LIN {X 0,Y 105.303,Z 769.102,A -85,B 0,C 180,E1 -26364.249,E2 -26364.249} C_VEL
LIN {X 0,Y 105.299,Z 772.199,A -85,B 0,C 180,E1 -26369.995,E2 -26369.995} C_VEL
LIN {X 0,Y 105.168,Z 773.673,A -85,B 0,C 180,E1 -26373.826,E2 -26373.826} C_VEL
LIN {X 0,Y 105.345,Z 774.732,A -85,B 0,C 180,E1 -26377.662,E2 -26377.662} C_VEL
LIN {X 0,Y 106.79,Z 775.648,A -85,B 0,C 180,E1 -26385.257,E2 -26385.257} C_VEL
LIN {X 0,Y 109.908,Z 775.104,A -85,B 0,C 180,E1 -26392.555,E2 -26392.555} C_VEL
LIN {X 0,Y 112.231,Z 774.277,A -85,B 0,C 180,E1 -26395.992,E2 -26395.992} C_VEL
LIN {X 0,Y 118.036,Z 771.438,A -85,B 0,C 180,E1 -26402.397,E2 -26402.397} C_VEL
LIN {X 0,Y 125.236,Z 766.969,A -85,B 0,C 180,E1 -26408.216,E2 -26408.216} C_VEL
LIN {X 0,Y 131.258,Z 762.539,A -85,B 0,C 180,E1 -26412.006,E2 -26412.006} C_VEL
LIN {X 0,Y 139.26,Z 755.845,A -85,B 0,C 180,E1 -26415.978,E2 -26415.978} C_VEL
LIN {X 0,Y 146.598,Z 748.7,A -85,B 0,C 180,E1 -26419.025,E2 -26419.025} C_VEL
LIN {X 0,Y 154.378,Z 739.924,A -85,B 0,C 180,E1 -26421.742,E2 -26421.742} C_VEL
LIN {X 0,Y 161.875,Z 729.959,A -85,B 0,C 180,E1 -26423.955,E2 -26423.955} C_VEL
LIN {X 0,Y 168.922,Z 718.713,A -85,B 0,C 180,E1 -26425.775,E2 -26425.775} C_VEL
LIN {X 0,Y 174.757,Z 707.532,A -85,B 0,C 180,E1 -26427.081,E2 -26427.081} C_VEL
LIN {X 0,Y 175.208,Z 706.525,A -85,B 0,C 180,E1 -26427.178,E2 -26427.178} C_VEL
LIN {X 0,Y 176.538,Z 703.106,A -85,B 0,C 180,E1 -26427.707,E2 -26427.707} C_VEL
LIN {X 0,Y 179.141,Z 692.574,A -85,B 0,C 180,E1 -26430.31,E2 -26430.31} C_VEL
LIN {X 0,Y 180.193,Z 688.973,A -85,B 0,C 180,E1 -26430.72,E2 -26430.72} C_VEL
LIN {X 0,Y 183.852,Z 675.631,A -85,B 0,C 180,E1 -26431.326,E2 -26431.326} C_VEL
LIN {X 0,Y 185.48,Z 666.767,A -85,B 0,C 180,E1 -26431.645,E2 -26431.645} C_VEL
LIN {X 0,Y 184.736,Z 662.719,A -85,B 0,C 180,E1 -26434.358,E2 -26434.358} C_VEL
LIN {X 0,Y 184.119,Z 659.45,A -85,B 0,C 180,E1 -26438.256,E2 -26438.256} C_VEL
LIN {X 0,Y 184.228,Z 658.963,A -85,B 0,C 180,E1 -26442.487,E2 -26442.487} C_VEL
LIN {X 0,Y 185.103,Z 661.189,A -85,B 0,C 180,E1 -26446.452,E2 -26446.452} C_VEL
LIN {X 0,Y 185.885,Z 663.628,A -85,B 0,C 180,E1 -26448.675,E2 -26448.675} C_VEL
LIN {X 0,Y 183.18,Z 677.331,A -85,B 0,C 180,E1 -26449.199,E2 -26449.199} C_VEL
LIN {X 0,Y 179.514,Z 689.858,A -85,B 0,C 180,E1 -26449.939,E2 -26449.939} C_VEL
LIN {X 0,Y 174.557,Z 702.362,A -85,B 0,C 180,E1 -26451.004,E2 -26451.004} C_VEL
LIN {X 0,Y 169.094,Z 713.244,A -85,B 0,C 180,E1 -26452.244,E2 -26452.244} C_VEL
LIN {X 0,Y 162.575,Z 723.845,A -85,B 0,C 180,E1 -26453.826,E2 -26453.826} C_VEL
LIN {X 0,Y 154.993,Z 734.01,A -85,B 0,C 180,E1 -26455.944,E2 -26455.944} C_VEL
LIN {X 0,Y 147.643,Z 742.315,A -85,B 0,C 180,E1 -26458.279,E2 -26458.279} C_VEL
LIN {X 0,Y 139.13,Z 750.499,A -85,B 0,C 180,E1 -26461.412,E2 -26461.412} C_VEL
LIN {X 0,Y 130.939,Z 757.072,A -85,B 0,C 180,E1 -26465.062,E2 -26465.062} C_VEL
LIN {X 0,Y 122.214,Z 762.916,A -85,B 0,C 180,E1 -26469.932,E2 -26469.932} C_VEL
LIN {X 0,Y 116.026,Z 766.288,A -85,B 0,C 180,E1 -26474.287,E2 -26474.287} C_VEL
LIN {X 0,Y 111.192,Z 768.427,A -85,B 0,C 180,E1 -26478.56,E2 -26478.56} C_VEL
LIN {X 0,Y 106.98,Z 769.842,A -85,B 0,C 180,E1 -26483.212,E2 -26483.212} C_VEL
LIN {X 0,Y 103.362,Z 770.554,A -85,B 0,C 180,E1 -26488.419,E2 -26488.419} C_VEL
LIN {X 0,Y 100.652,Z 770.454,A -85,B 0,C 180,E1 -26493.956,E2 -26493.956} C_VEL
LIN {X 0,Y 98.728,Z 769.526,A -85,B 0,C 180,E1 -26499.839,E2 -26499.839} C_VEL
LIN {X 0,Y 97.648,Z 767.699,A -85,B 0,C 180,E1 -26506.029,E2 -26506.029} C_VEL
LIN {X 0,Y 97.544,Z 764.862,A -85,B 0,C 180,E1 -26512.42,E2 -26512.42} C_VEL
LIN {X 0,Y 98.341,Z 760.757,A -85,B 0,C 180,E1 -26519.043,E2 -26519.043} C_VEL
LIN {X 0,Y 100.087,Z 755.004,A -85,B 0,C 180,E1 -26525.897,E2 -26525.897} C_VEL
LIN {X 0,Y 102.312,Z 748.886,A -85,B 0,C 180,E1 -26531.427,E2 -26531.427} C_VEL
LIN {X 0,Y 105.063,Z 741.752,A -85,B 0,C 180,E1 -26536.466,E2 -26536.466} C_VEL
LIN {X 0,Y 108.553,Z 733.143,A -85,B 0,C 180,E1 -26541.16,E2 -26541.16} C_VEL
LIN {X 0,Y 112.175,Z 723.535,A -85,B 0,C 180,E1 -26545.211,E2 -26545.211} C_VEL
LIN {X 0,Y 116.013,Z 712.64,A -85,B 0,C 180,E1 -26548.703,E2 -26548.703} C_VEL
LIN {X 0,Y 119.515,Z 700.829,A -85,B 0,C 180,E1 -26551.54,E2 -26551.54} C_VEL
LIN {X 0,Y 122.584,Z 688.566,A -85,B 0,C 180,E1 -26553.703,E2 -26553.703} C_VEL
LIN {X 0,Y 125.058,Z 675.36,A -85,B 0,C 180,E1 -26555.345,E2 -26555.345} C_VEL
LIN {X 0,Y 126.899,Z 661.316,A -85,B 0,C 180,E1 -26556.426,E2 -26556.426} C_VEL
LIN {X 0,Y 130.052,Z 624.131,A -85,B 0,C 180,E1 -26558.464,E2 -26558.464} C_VEL
LIN {X 0,Y 123.711,Z 608.885,A -85,B 0,C 180,E1 -26561.983,E2 -26561.983} C_VEL
LIN {X 0,Y 115.972,Z 594.893,A -85,B 0,C 180,E1 -26566.547,E2 -26566.547} C_VEL
LIN {X 0,Y 110.04,Z 585.76,A -85,B 0,C 180,E1 -26570.479,E2 -26570.479} C_VEL
LIN {X 0,Y 107.393,Z 581.803,A -85,B 0,C 180,E1 -26572.446,E2 -26572.446} C_VEL
LIN {X 0,Y 104.798,Z 578.322,A -85,B 0,C 180,E1 -26574.502,E2 -26574.502} C_VEL
LIN {X 0,Y 104.228,Z 577.151,A -85,B 0,C 180,E1 -26575.032,E2 -26575.032} C_VEL
LIN {X 0,Y 102,Z 575.216,A -85,B 0,C 180,E1 -26576.806,E2 -26576.806} C_VEL
LIN {X 0,Y 100.845,Z 572.761,A -85,B 0,C 180,E1 -26577.978,E2 -26577.978} C_VEL
LIN {X 0,Y 100.663,Z 571.949,A -85,B 0,C 180,E1 -26578.344,E2 -26578.344} C_VEL
LIN {X 0,Y 100.666,Z 571.937,A -85,B 0,C 180,E1 -26583.96,E2 -26583.96} C_VEL
LIN {X 0,Y 100.643,Z 571.931,A -85,B 0,C 180,E1 -26589.816,E2 -26589.816} C_VEL
LIN {X 0,Y 100.652,Z 571.948,A -85,B 0,C 180,E1 -26595.716,E2 -26595.716} C_VEL
LIN {X 0,Y 100.631,Z 571.925,A -85,B 0,C 180,E1 -26601.059,E2 -26601.059} C_VEL
LIN {X 0,Y 100.695,Z 571.94,A -85,B 0,C 180,E1 -26606.891,E2 -26606.891} C_VEL
LIN {X 0,Y 100.794,Z 571.925,A -85,B 0,C 180,E1 -26615.271,E2 -26615.271} C_VEL
LIN {X 0,Y 100.816,Z 571.915,A -85,B 0,C 180,E1 -26619.603,E2 -26619.603} C_VEL
LIN {X 0,Y 101.168,Z 571.883,A -85,B 0,C 180,E1 -26627.973,E2 -26627.973} C_VEL
LIN {X 0,Y 101.251,Z 571.851,A -85,B 0,C 180,E1 -26632.022,E2 -26632.022} C_VEL
LIN {X 0,Y 101.876,Z 571.793,A -85,B 0,C 180,E1 -26640.002,E2 -26640.002} C_VEL
LIN {X 0,Y 101.285,Z 571.868,A -85,B 0,C 180,E1 -26647.979,E2 -26647.979} C_VEL
LIN {X 0,Y 101.123,Z 571.872,A -85,B 0,C 180,E1 -26653.324,E2 -26653.324} C_VEL
LIN {X 0,Y 100.824,Z 571.887,A -85,B 0,C 180,E1 -26661.334,E2 -26661.334} C_VEL
LIN {X 0,Y 101.671,Z 574.415,A -85,B 0,C 180,E1 -26662.347,E2 -26662.347} C_VEL
LIN {X 0,Y 103.856,Z 576.845,A -85,B 0,C 180,E1 -26664.223,E2 -26664.223} C_VEL
LIN {X 0,Y 106.376,Z 580.87,A -85,B 0,C 180,E1 -26666.354,E2 -26666.354} C_VEL
LIN {X 0,Y 107.782,Z 582.765,A -85,B 0,C 180,E1 -26667.423,E2 -26667.423} C_VEL
LIN {X 0,Y 112.491,Z 589.94,A -85,B 0,C 180,E1 -26670.767,E2 -26670.767} C_VEL
LIN {X 0,Y 118.61,Z 600.466,A -85,B 0,C 180,E1 -26674.709,E2 -26674.709} C_VEL
LIN {X 0,Y 122.562,Z 609.707,A -85,B 0,C 180,E1 -26677.165,E2 -26677.165} C_VEL
LIN {X 0,Y 126.766,Z 621.513,A -85,B 0,C 180,E1 -26679.728,E2 -26679.728} C_VEL
LIN {X 0,Y 129.782,Z 631.148,A -85,B 0,C 180,E1 -26681.535,E2 -26681.535} C_VEL
LIN {X 0,Y 126.025,Z 673.787,A -85,B 0,C 180,E1 -26683.961,E2 -26683.961} C_VEL
LIN {X 0,Y 123.841,Z 687.25,A -85,B 0,C 180,E1 -26685.241,E2 -26685.241} C_VEL
LIN {X 0,Y 121.065,Z 699.593,A -85,B 0,C 180,E1 -26686.986,E2 -26686.986} C_VEL
LIN {X 0,Y 117.605,Z 711.948,A -85,B 0,C 180,E1 -26689.461,E2 -26689.461} C_VEL
LIN {X 0,Y 113.967,Z 723.108,A -85,B 0,C 180,E1 -26692.479,E2 -26692.479} C_VEL
LIN {X 0,Y 110.055,Z 733.645,A -85,B 0,C 180,E1 -26696.283,E2 -26696.283} C_VEL
LIN {X 0,Y 106.01,Z 743.969,A -85,B 0,C 180,E1 -26701.267,E2 -26701.267} C_VEL
LIN {X 0,Y 102.656,Z 752.512,A -85,B 0,C 180,E1 -26706.812,E2 -26706.812} C_VEL
LIN {X 0,Y 100.226,Z 759.339,A -85,B 0,C 180,E1 -26712.656,E2 -26712.656} C_VEL
LIN {X 0,Y 98.654,Z 765.567,A -85,B 0,C 180,E1 -26719.735,E2 -26719.735} C_VEL
LIN {X 0,Y 98.19,Z 769.554,A -85,B 0,C 180,E1 -26725.89,E2 -26725.89} C_VEL
LIN {X 0,Y 98.234,Z 771.574,A -85,B 0,C 180,E1 -26729.994,E2 -26729.994} C_VEL
LIN {X 0,Y 98.094,Z 773.12,A -85,B 0,C 180,E1 -26734.103,E2 -26734.103} C_VEL
LIN {X 0,Y 98.897,Z 775.038,A -85,B 0,C 180,E1 -26742.303,E2 -26742.303} C_VEL
LIN {X 0,Y 101.407,Z 775.387,A -85,B 0,C 180,E1 -26750.269,E2 -26750.269} C_VEL
LIN {X 0,Y 105.888,Z 774.285,A -85,B 0,C 180,E1 -26757.678,E2 -26757.678} C_VEL
LIN {X 0,Y 112.1,Z 771.687,A -85,B 0,C 180,E1 -26764.343,E2 -26764.343} C_VEL
LIN {X 0,Y 119.646,Z 767.467,A -85,B 0,C 180,E1 -26770.245,E2 -26770.245} C_VEL
LIN {X 0,Y 126.112,Z 763.193,A -85,B 0,C 180,E1 -26774.148,E2 -26774.148} C_VEL
LIN {X 0,Y 134.473,Z 756.819,A -85,B 0,C 180,E1 -26778.131,E2 -26778.131} C_VEL
LIN {X 0,Y 142.121,Z 749.947,A -85,B 0,C 180,E1 -26781.149,E2 -26781.149} C_VEL
LIN {X 0,Y 150.176,Z 741.472,A -85,B 0,C 180,E1 -26783.823,E2 -26783.823} C_VEL
LIN {X 0,Y 157.178,Z 732.942,A -85,B 0,C 180,E1 -26785.805,E2 -26785.805} C_VEL
LIN {X 0,Y 164.413,Z 722.56,A -85,B 0,C 180,E1 -26787.583,E2 -26787.583} C_VEL
LIN {X 0,Y 171.098,Z 710.87,A -85,B 0,C 180,E1 -26789.025,E2 -26789.025} C_VEL
LIN {X 0,Y 176.407,Z 699.321,A -85,B 0,C 180,E1 -26790.048,E2 -26790.048} C_VEL
LIN {X 0,Y 180.193,Z 688.973,A -85,B 0,C 180,E1 -26790.72,E2 -26790.72} C_VEL
LIN {X 0,Y 182.064,Z 682.31,A -85,B 0,C 180,E1 -26791.231,E2 -26791.231} C_VEL
LIN {X 0,Y 183.034,Z 677.264,A -85,B 0,C 180,E1 -26791.947,E2 -26791.947} C_VEL
LIN {X 0,Y 183.418,Z 673.974,A -85,B 0,C 180,E1 -26792.699,E2 -26792.699} C_VEL
LIN {X 0,Y 183.499,Z 671.379,A -85,B 0,C 180,E1 -26793.666,E2 -26793.666} C_VEL
LIN {X 0,Y 183.46,Z 670.748,A -85,B 0,C 180,E1 -26794.038,E2 -26794.038} C_VEL
LIN {X 0,Y 183.185,Z 668.656,A -85,B 0,C 180,E1 -26795.704,E2 -26795.704} C_VEL
LIN {X 0,Y 182.935,Z 666.303,A -85,B 0,C 180,E1 -26798.908,E2 -26798.908} C_VEL
LIN {X 0,Y 183.127,Z 666.057,A -85,B 0,C 180,E1 -26802.726,E2 -26802.726} C_VEL
LIN {X 0,Y 183.726,Z 668.003,A -85,B 0,C 180,E1 -26805.967,E2 -26805.967} C_VEL
LIN {X 0,Y 183.867,Z 668.892,A -85,B 0,C 180,E1 -26806.677,E2 -26806.677} C_VEL
LIN {X 0,Y 180.525,Z 682.697,A -85,B 0,C 180,E1 -26807.255,E2 -26807.255} C_VEL
LIN {X 0,Y 176.457,Z 694.617,A -85,B 0,C 180,E1 -26808.019,E2 -26808.019} C_VEL
LIN {X 0,Y 170.967,Z 706.812,A -85,B 0,C 180,E1 -26809.11,E2 -26809.11} C_VEL
LIN {X 0,Y 164.778,Z 717.747,A -85,B 0,C 180,E1 -26810.431,E2 -26810.431} C_VEL
LIN {X 0,Y 158.017,Z 727.658,A -85,B 0,C 180,E1 -26812.016,E2 -26812.016} C_VEL
LIN {X 0,Y 150.126,Z 737.27,A -85,B 0,C 180,E1 -26814.098,E2 -26814.098} C_VEL
LIN {X 0,Y 142.587,Z 745.015,A -85,B 0,C 180,E1 -26816.403,E2 -26816.403} C_VEL
LIN {X 0,Y 133.524,Z 752.841,A -85,B 0,C 180,E1 -26819.617,E2 -26819.617} C_VEL
LIN {X 0,Y 125.3,Z 758.814,A -85,B 0,C 180,E1 -26823.214,E2 -26823.214} C_VEL
LIN {X 0,Y 116.21,Z 764.188,A -85,B 0,C 180,E1 -26828.147,E2 -26828.147} C_VEL
LIN {X 0,Y 108.475,Z 767.805,A -85,B 0,C 180,E1 -26833.654,E2 -26833.654} C_VEL
LIN {X 0,Y 101.706,Z 770.024,A -85,B 0,C 180,E1 -26840.21,E2 -26840.21} C_VEL
LIN {X 0,Y 97.606,Z 770.773,A -85,B 0,C 180,E1 -26845.594,E2 -26845.594} C_VEL
LIN {X 0,Y 93.331,Z 770.407,A -85,B 0,C 180,E1 -26854.085,E2 -26854.085} C_VEL
LIN {X 0,Y 91.54,Z 769.325,A -85,B 0,C 180,E1 -26859.858,E2 -26859.858} C_VEL
LIN {X 0,Y 90.414,Z 766.441,A -85,B 0,C 180,E1 -26868.538,E2 -26868.538} C_VEL
LIN {X 0,Y 90.943,Z 761.922,A -85,B 0,C 180,E1 -26877.259,E2 -26877.259} C_VEL
LIN {X 0,Y 92.41,Z 756.802,A -85,B 0,C 180,E1 -26884.25,E2 -26884.25} C_VEL
LIN {X 0,Y 94.536,Z 750.833,A -85,B 0,C 180,E1 -26890.464,E2 -26890.464} C_VEL
LIN {X 0,Y 97.596,Z 743.305,A -85,B 0,C 180,E1 -26896.471,E2 -26896.471} C_VEL
LIN {X 0,Y 101.499,Z 734.024,A -85,B 0,C 180,E1 -26902.046,E2 -26902.046} C_VEL
LIN {X 0,Y 105.598,Z 723.772,A -85,B 0,C 180,E1 -26906.639,E2 -26906.639} C_VEL
LIN {X 0,Y 109.721,Z 712.599,A -85,B 0,C 180,E1 -26910.377,E2 -26910.377} C_VEL
LIN {X 0,Y 113.283,Z 701.181,A -85,B 0,C 180,E1 -26913.223,E2 -26913.223} C_VEL
LIN {X 0,Y 116.772,Z 687.915,A -85,B 0,C 180,E1 -26915.617,E2 -26915.617} C_VEL
LIN {X 0,Y 119.258,Z 674.646,A -85,B 0,C 180,E1 -26917.282,E2 -26917.282} C_VEL
LIN {X 0,Y 121.047,Z 661.623,A -85,B 0,C 180,E1 -26918.288,E2 -26918.288} C_VEL
LIN {X 0,Y 124.269,Z 626.1,A -85,B 0,C 180,E1 -26920.271,E2 -26920.271} C_VEL
LIN {X 0,Y 118.738,Z 612.717,A -85,B 0,C 180,E1 -26923.581,E2 -26923.581} C_VEL
LIN {X 0,Y 111.803,Z 599.793,A -85,B 0,C 180,E1 -26928.036,E2 -26928.036} C_VEL
LIN {X 0,Y 106.071,Z 590.815,A -85,B 0,C 180,E1 -26932.154,E2 -26932.154} C_VEL
LIN {X 0,Y 102.725,Z 585.931,A -85,B 0,C 180,E1 -26934.902,E2 -26934.902} C_VEL
LIN {X 0,Y 100.659,Z 582.889,A -85,B 0,C 180,E1 -26936.715,E2 -26936.715} C_VEL
LIN {X 0,Y 98.196,Z 579.989,A -85,B 0,C 180,E1 -26938.969,E2 -26938.969} C_VEL
LIN {X 0,Y 97.32,Z 578.208,A -85,B 0,C 180,E1 -26939.94,E2 -26939.94} C_VEL
LIN {X 0,Y 94.941,Z 576.16,A -85,B 0,C 180,E1 -26942.331,E2 -26942.331} C_VEL
LIN {X 0,Y 93.694,Z 573.326,A -85,B 0,C 180,E1 -26944.003,E2 -26944.003} C_VEL
LIN {X 0,Y 93.595,Z 572.819,A -85,B 0,C 180,E1 -26944.315,E2 -26944.315} C_VEL
LIN {X 0,Y 93.537,Z 572.819,A -85,B 0,C 180,E1 -26952.557,E2 -26952.557} C_VEL
LIN {X 0,Y 93.54,Z 572.813,A -85,B 0,C 180,E1 -26958.715,E2 -26958.715} C_VEL
LIN {X 0,Y 93.592,Z 572.828,A -85,B 0,C 180,E1 -26965.701,E2 -26965.701} C_VEL
LIN {X 0,Y 93.675,Z 572.802,A -85,B 0,C 180,E1 -26974.211,E2 -26974.211} C_VEL
LIN {X 0,Y 93.696,Z 572.811,A -85,B 0,C 180,E1 -26977.976,E2 -26977.976} C_VEL
LIN {X 0,Y 94.077,Z 572.764,A -85,B 0,C 180,E1 -26987.051,E2 -26987.051} C_VEL
LIN {X 0,Y 94.185,Z 572.734,A -85,B 0,C 180,E1 -26991.419,E2 -26991.419} C_VEL
LIN {X 0,Y 94.801,Z 572.674,A -85,B 0,C 180,E1 -27000.002,E2 -27000.002} C_VEL
LIN {X 0,Y 94.218,Z 572.75,A -85,B 0,C 180,E1 -27008.582,E2 -27008.582} C_VEL
LIN {X 0,Y 94.044,Z 572.754,A -85,B 0,C 180,E1 -27013.689,E2 -27013.689} C_VEL
LIN {X 0,Y 93.907,Z 572.785,A -85,B 0,C 180,E1 -27015.639,E2 -27015.639} C_VEL
LIN {X 0,Y 94.721,Z 575.446,A -85,B 0,C 180,E1 -27016.858,E2 -27016.858} C_VEL
LIN {X 0,Y 96.625,Z 577.643,A -85,B 0,C 180,E1 -27018.882,E2 -27018.882} C_VEL
LIN {X 0,Y 97.639,Z 578.51,A -85,B 0,C 180,E1 -27019.857,E2 -27019.857} C_VEL
LIN {X 0,Y 99.718,Z 581.799,A -85,B 0,C 180,E1 -27021.942,E2 -27021.942} C_VEL
LIN {X 0,Y 100.982,Z 583.43,A -85,B 0,C 180,E1 -27023.083,E2 -27023.083} C_VEL
LIN {X 0,Y 103.649,Z 587.259,A -85,B 0,C 180,E1 -27025.423,E2 -27025.423} C_VEL
LIN {X 0,Y 109.031,Z 596,A -85,B 0,C 180,E1 -27029.64,E2 -27029.64} C_VEL
LIN {X 0,Y 114.357,Z 605.405,A -85,B 0,C 180,E1 -27033.293,E2 -27033.293} C_VEL
LIN {X 0,Y 118.618,Z 616.25,A -85,B 0,C 180,E1 -27036.217,E2 -27036.217} C_VEL
LIN {X 0,Y 122.728,Z 628.647,A -85,B 0,C 180,E1 -27038.914,E2 -27038.914} C_VEL
LIN {X 0,Y 123.981,Z 632.936,A -85,B 0,C 180,E1 -27039.732,E2 -27039.732} C_VEL
LIN {X 0,Y 120.183,Z 673.625,A -85,B 0,C 180,E1 -27042.097,E2 -27042.097} C_VEL
LIN {X 0,Y 117.913,Z 687.04,A -85,B 0,C 180,E1 -27043.407,E2 -27043.407} C_VEL
LIN {X 0,Y 114.895,Z 699.847,A -85,B 0,C 180,E1 -27045.29,E2 -27045.29} C_VEL
LIN {X 0,Y 111.273,Z 712.077,A -85,B 0,C 180,E1 -27047.843,E2 -27047.843} C_VEL
LIN {X 0,Y 107.478,Z 723.156,A -85,B 0,C 180,E1 -27050.989,E2 -27050.989} C_VEL
LIN {X 0,Y 103.561,Z 733.174,A -85,B 0,C 180,E1 -27054.779,E2 -27054.779} C_VEL
LIN {X 0,Y 99.795,Z 742.237,A -85,B 0,C 180,E1 -27059.291,E2 -27059.291} C_VEL
LIN {X 0,Y 96.156,Z 751.117,A -85,B 0,C 180,E1 -27065.142,E2 -27065.142} C_VEL
LIN {X 0,Y 93.433,Z 758.164,A -85,B 0,C 180,E1 -27071.35,E2 -27071.35} C_VEL
LIN {X 0,Y 92.05,Z 762.964,A -85,B 0,C 180,E1 -27076.753,E2 -27076.753} C_VEL
LIN {X 0,Y 91.215,Z 767.526,A -85,B 0,C 180,E1 -27083.357,E2 -27083.357} C_VEL
LIN {X 0,Y 91.159,Z 770.934,A -85,B 0,C 180,E1 -27089.994,E2 -27089.994} C_VEL
LIN {X 0,Y 91.033,Z 772.568,A -85,B 0,C 180,E1 -27094.421,E2 -27094.421} C_VEL
LIN {X 0,Y 91.972,Z 774.634,A -85,B 0,C 180,E1 -27103.246,E2 -27103.246} C_VEL
LIN {X 0,Y 94.744,Z 775.214,A -85,B 0,C 180,E1 -27111.764,E2 -27111.764} C_VEL
LIN {X 0,Y 99.651,Z 774.282,A -85,B 0,C 180,E1 -27119.576,E2 -27119.576} C_VEL
LIN {X 0,Y 106.313,Z 771.897,A -85,B 0,C 180,E1 -27126.503,E2 -27126.503} C_VEL
LIN {X 0,Y 113.657,Z 768.333,A -85,B 0,C 180,E1 -27132.093,E2 -27132.093} C_VEL
LIN {X 0,Y 121.159,Z 763.868,A -85,B 0,C 180,E1 -27136.468,E2 -27136.468} C_VEL
LIN {X 0,Y 128.634,Z 758.696,A -85,B 0,C 180,E1 -27139.891,E2 -27139.891} C_VEL
LIN {X 0,Y 135.135,Z 753.511,A -85,B 0,C 180,E1 -27142.47,E2 -27142.47} C_VEL
LIN {X 0,Y 143.375,Z 745.974,A -85,B 0,C 180,E1 -27145.183,E2 -27145.183} C_VEL
LIN {X 0,Y 151.932,Z 736.663,A -85,B 0,C 180,E1 -27147.579,E2 -27147.579} C_VEL
LIN {X 0,Y 159.326,Z 727.15,A -85,B 0,C 180,E1 -27149.327,E2 -27149.327} C_VEL
LIN {X 0,Y 166.141,Z 716.698,A -85,B 0,C 180,E1 -27150.739,E2 -27150.739} C_VEL
LIN {X 0,Y 172.313,Z 705.095,A -85,B 0,C 180,E1 -27151.877,E2 -27151.877} C_VEL
LIN {X 0,Y 177.442,Z 692.926,A -85,B 0,C 180,E1 -27152.736,E2 -27152.736} C_VEL
LIN {X 0,Y 181.554,Z 679.917,A -85,B 0,C 180,E1 -27153.348,E2 -27153.348} C_VEL
LIN {X 0,Y 183.521,Z 671.13,A -85,B 0,C 180,E1 -27153.73,E2 -27153.73} C_VEL
LIN {X 0,Y 183.46,Z 670.748,A -85,B 0,C 180,E1 -27154.038,E2 -27154.038} C_VEL
LIN {X 0,Y 183.232,Z 669.591,A -85,B 0,C 180,E1 -27155.204,E2 -27155.204} C_VEL
LIN {X 0,Y 182.925,Z 669.204,A -85,B 0,C 180,E1 -27156.423,E2 -27156.423} C_VEL
LIN {X 0,Y 182.431,Z 669.68,A -85,B 0,C 180,E1 -27158.284,E2 -27158.284} C_VEL
LIN {X 0,Y 181.8,Z 673.828,A -85,B 0,C 180,E1 -27163.994,E2 -27163.994} C_VEL
LIN {X 0,Y 181.888,Z 674.163,A -85,B 0,C 180,E1 -27164.65,E2 -27164.65} C_VEL
LIN {X 0,Y 178.077,Z 687.429,A -85,B 0,C 180,E1 -27165.248,E2 -27165.248} C_VEL
LIN {X 0,Y 173.312,Z 699.666,A -85,B 0,C 180,E1 -27166.1,E2 -27166.1} C_VEL
LIN {X 0,Y 167.586,Z 711.035,A -85,B 0,C 180,E1 -27167.151,E2 -27167.151} C_VEL
LIN {X 0,Y 160.432,Z 722.36,A -85,B 0,C 180,E1 -27168.552,E2 -27168.552} C_VEL
LIN {X 0,Y 152.361,Z 732.83,A -85,B 0,C 180,E1 -27170.366,E2 -27170.366} C_VEL
LIN {X 0,Y 143.363,Z 742.363,A -85,B 0,C 180,E1 -27172.713,E2 -27172.713} C_VEL
LIN {X 0,Y 133.917,Z 750.714,A -85,B 0,C 180,E1 -27175.59,E2 -27175.59} C_VEL
LIN {X 0,Y 126.551,Z 756.163,A -85,B 0,C 180,E1 -27178.27,E2 -27178.27} C_VEL
LIN {X 0,Y 119.496,Z 760.625,A -85,B 0,C 180,E1 -27181.308,E2 -27181.308} C_VEL
LIN {X 0,Y 110.327,Z 765.42,A -85,B 0,C 180,E1 -27186.165,E2 -27186.165} C_VEL
LIN {X 0,Y 102.121,Z 768.687,A -85,B 0,C 180,E1 -27191.913,E2 -27191.913} C_VEL
LIN {X 0,Y 95.925,Z 770.391,A -85,B 0,C 180,E1 -27197.761,E2 -27197.761} C_VEL
LIN {X 0,Y 91.653,Z 771.015,A -85,B 0,C 180,E1 -27203.066,E2 -27203.066} C_VEL
LIN {X 0,Y 88.244,Z 770.918,A -85,B 0,C 180,E1 -27208.843,E2 -27208.843} C_VEL
LIN {X 0,Y 85.729,Z 770.107,A -85,B 0,C 180,E1 -27215.017,E2 -27215.017} C_VEL
LIN {X 0,Y 83.928,Z 768.41,A -85,B 0,C 180,E1 -27222.056,E2 -27222.056} C_VEL
LIN {X 0,Y 83.314,Z 765.764,A -85,B 0,C 180,E1 -27229.389,E2 -27229.389} C_VEL
LIN {X 0,Y 83.787,Z 761.936,A -85,B 0,C 180,E1 -27237.008,E2 -27237.008} C_VEL
LIN {X 0,Y 85.381,Z 756.557,A -85,B 0,C 180,E1 -27244.877,E2 -27244.877} C_VEL
LIN {X 0,Y 87.541,Z 750.8,A -85,B 0,C 180,E1 -27251.276,E2 -27251.276} C_VEL
LIN {X 0,Y 90.724,Z 743.376,A -85,B 0,C 180,E1 -27257.591,E2 -27257.591} C_VEL
LIN {X 0,Y 94.523,Z 734.874,A -85,B 0,C 180,E1 -27263.067,E2 -27263.067} C_VEL
LIN {X 0,Y 98.472,Z 725.496,A -85,B 0,C 180,E1 -27267.632,E2 -27267.632} C_VEL
LIN {X 0,Y 102.6,Z 714.998,A -85,B 0,C 180,E1 -27271.478,E2 -27271.478} C_VEL
LIN {X 0,Y 106.341,Z 704.212,A -85,B 0,C 180,E1 -27274.452,E2 -27274.452} C_VEL
LIN {X 0,Y 109.756,Z 692.262,A -85,B 0,C 180,E1 -27276.901,E2 -27276.901} C_VEL
LIN {X 0,Y 112.679,Z 679.249,A -85,B 0,C 180,E1 -27278.778,E2 -27278.778} C_VEL
LIN {X 0,Y 114.73,Z 666.76,A -85,B 0,C 180,E1 -27279.973,E2 -27279.973} C_VEL
LIN {X 0,Y 118.528,Z 628.194,A -85,B 0,C 180,E1 -27282.205,E2 -27282.205} C_VEL
LIN {X 0,Y 114.105,Z 617.066,A -85,B 0,C 180,E1 -27285.155,E2 -27285.155} C_VEL
LIN {X 0,Y 107.451,Z 604.295,A -85,B 0,C 180,E1 -27289.791,E2 -27289.791} C_VEL
LIN {X 0,Y 101.928,Z 595.485,A -85,B 0,C 180,E1 -27294.189,E2 -27294.189} C_VEL
LIN {X 0,Y 97.589,Z 588.871,A -85,B 0,C 180,E1 -27298.146,E2 -27298.146} C_VEL
LIN {X 0,Y 94.902,Z 585.392,A -85,B 0,C 180,E1 -27300.88,E2 -27300.88} C_VEL
LIN {X 0,Y 94.09,Z 584.155,A -85,B 0,C 180,E1 -27301.802,E2 -27301.802} C_VEL
LIN {X 0,Y 91.705,Z 581.35,A -85,B 0,C 180,E1 -27304.605,E2 -27304.605} C_VEL
LIN {X 0,Y 90.646,Z 579.321,A -85,B 0,C 180,E1 -27306.087,E2 -27306.087} C_VEL
LIN {X 0,Y 88.114,Z 577.476,A -85,B 0,C 180,E1 -27309.386,E2 -27309.386} C_VEL
LIN {X 0,Y 86.79,Z 575.014,A -85,B 0,C 180,E1 -27311.712,E2 -27311.712} C_VEL
LIN {X 0,Y 86.501,Z 573.694,A -85,B 0,C 180,E1 -27312.513,E2 -27312.513} C_VEL
LIN {X 0,Y 86.461,Z 573.69,A -85,B 0,C 180,E1 -27319.441,E2 -27319.441} C_VEL
LIN {X 0,Y 86.535,Z 573.706,A -85,B 0,C 180,E1 -27325.357,E2 -27325.357} C_VEL
LIN {X 0,Y 86.589,Z 573.675,A -85,B 0,C 180,E1 -27333.243,E2 -27333.243} C_VEL
LIN {X 0,Y 86.638,Z 573.666,A -85,B 0,C 180,E1 -27341.069,E2 -27341.069} C_VEL
LIN {X 0,Y 86.94,Z 573.643,A -85,B 0,C 180,E1 -27345.968,E2 -27345.968} C_VEL
LIN {X 0,Y 87.094,Z 573.622,A -85,B 0,C 180,E1 -27350.715,E2 -27350.715} C_VEL
LIN {X 0,Y 87.728,Z 573.555,A -85,B 0,C 180,E1 -27360.002,E2 -27360.002} C_VEL
LIN {X 0,Y 87.156,Z 573.634,A -85,B 0,C 180,E1 -27367.969,E2 -27367.969} C_VEL
LIN {X 0,Y 88.044,Z 576.363,A -85,B 0,C 180,E1 -27369.768,E2 -27369.768} C_VEL
LIN {X 0,Y 89.827,Z 578.433,A -85,B 0,C 180,E1 -27372.346,E2 -27372.346} C_VEL
LIN {X 0,Y 91.023,Z 579.404,A -85,B 0,C 180,E1 -27373.868,E2 -27373.868} C_VEL
LIN {X 0,Y 92.772,Z 582.639,A -85,B 0,C 180,E1 -27376.224,E2 -27376.224} C_VEL
LIN {X 0,Y 94.81,Z 584.857,A -85,B 0,C 180,E1 -27378.453,E2 -27378.453} C_VEL
LIN {X 0,Y 98.123,Z 589.876,A -85,B 0,C 180,E1 -27381.901,E2 -27381.901} C_VEL
LIN {X 0,Y 102.632,Z 596.778,A -85,B 0,C 180,E1 -27385.972,E2 -27385.972} C_VEL
LIN {X 0,Y 108.919,Z 607.942,A -85,B 0,C 180,E1 -27390.903,E2 -27390.903} C_VEL
LIN {X 0,Y 111.04,Z 612.609,A -85,B 0,C 180,E1 -27392.454,E2 -27392.454} C_VEL
LIN {X 0,Y 115.67,Z 625.814,A -85,B 0,C 180,E1 -27395.913,E2 -27395.913} C_VEL
LIN {X 0,Y 118.175,Z 634.265,A -85,B 0,C 180,E1 -27397.729,E2 -27397.729} C_VEL
LIN {X 0,Y 114.52,Z 672.517,A -85,B 0,C 180,E1 -27400.015,E2 -27400.015} C_VEL
LIN {X 0,Y 112.25,Z 685.699,A -85,B 0,C 180,E1 -27401.288,E2 -27401.288} C_VEL
LIN {X 0,Y 109.368,Z 697.803,A -85,B 0,C 180,E1 -27403.026,E2 -27403.026} C_VEL
LIN {X 0,Y 106.113,Z 708.916,A -85,B 0,C 180,E1 -27405.268,E2 -27405.268} C_VEL
LIN {X 0,Y 102.021,Z 720.507,A -85,B 0,C 180,E1 -27408.46,E2 -27408.46} C_VEL
LIN {X 0,Y 97.426,Z 731.977,A -85,B 0,C 180,E1 -27412.773,E2 -27412.773} C_VEL
LIN {X 0,Y 92.998,Z 742.121,A -85,B 0,C 180,E1 -27418.055,E2 -27418.055} C_VEL
LIN {X 0,Y 89.162,Z 750.981,A -85,B 0,C 180,E1 -27424.302,E2 -27424.302} C_VEL
LIN {X 0,Y 86.335,Z 758.012,A -85,B 0,C 180,E1 -27430.99,E2 -27430.99} C_VEL
LIN {X 0,Y 84.712,Z 763.62,A -85,B 0,C 180,E1 -27438.023,E2 -27438.023} C_VEL
LIN {X 0,Y 84.064,Z 767.959,A -85,B 0,C 180,E1 -27445.198,E2 -27445.198} C_VEL
LIN {X 0,Y 84.081,Z 770.21,A -85,B 0,C 180,E1 -27449.993,E2 -27449.993} C_VEL
LIN {X 0,Y 83.99,Z 771.973,A -85,B 0,C 180,E1 -27454.793,E2 -27454.793} C_VEL
LIN {X 0,Y 84.286,Z 773.296,A -85,B 0,C 180,E1 -27459.593,E2 -27459.593} C_VEL
LIN {X 0,Y 86.339,Z 774.774,A -85,B 0,C 180,E1 -27468.995,E2 -27468.995} C_VEL
LIN {X 0,Y 90.58,Z 774.815,A -85,B 0,C 180,E1 -27477.737,E2 -27477.737} C_VEL
LIN {X 0,Y 96.904,Z 773.373,A -85,B 0,C 180,E1 -27485.457,E2 -27485.457} C_VEL
LIN {X 0,Y 104.824,Z 770.435,A -85,B 0,C 180,E1 -27492.095,E2 -27492.095} C_VEL
LIN {X 0,Y 111.524,Z 767.186,A -85,B 0,C 180,E1 -27496.436,E2 -27496.436} C_VEL
LIN {X 0,Y 118.968,Z 762.982,A -85,B 0,C 180,E1 -27500.164,E2 -27500.164} C_VEL
LIN {X 0,Y 128.177,Z 756.73,A -85,B 0,C 180,E1 -27503.965,E2 -27503.965} C_VEL
LIN {X 0,Y 136.621,Z 749.976,A -85,B 0,C 180,E1 -27506.704,E2 -27506.704} C_VEL
LIN {X 0,Y 145.349,Z 741.67,A -85,B 0,C 180,E1 -27509.113,E2 -27509.113} C_VEL
LIN {X 0,Y 154.37,Z 731.44,A -85,B 0,C 180,E1 -27511.202,E2 -27511.202} C_VEL
LIN {X 0,Y 162.087,Z 720.869,A -85,B 0,C 180,E1 -27512.723,E2 -27512.723} C_VEL
LIN {X 0,Y 169.191,Z 708.839,A -85,B 0,C 180,E1 -27513.924,E2 -27513.924} C_VEL
LIN {X 0,Y 174.465,Z 697.676,A -85,B 0,C 180,E1 -27514.748,E2 -27514.748} C_VEL
LIN {X 0,Y 178.679,Z 686.35,A -85,B 0,C 180,E1 -27515.315,E2 -27515.315} C_VEL
LIN {X 0,Y 181.591,Z 675.797,A -85,B 0,C 180,E1 -27515.785,E2 -27515.785} C_VEL
LIN {X 0,Y 181.521,Z 673.212,A -85,B 0,C 180,E1 -27519.172,E2 -27519.172} C_VEL
LIN {X 0,Y 181.699,Z 673.013,A -85,B 0,C 180,E1 -27522.586,E2 -27522.586} C_VEL
LIN {X 0,Y 181.8,Z 673.828,A -85,B 0,C 180,E1 -27523.994,E2 -27523.994} C_VEL
LIN {X 0,Y 181.683,Z 674.658,A -85,B 0,C 180,E1 -27524.347,E2 -27524.347} C_VEL
LIN {X 0,Y 181.087,Z 677.099,A -85,B 0,C 180,E1 -27524.545,E2 -27524.545} C_VEL
LIN {X 0,Y 180.036,Z 680.704,A -85,B 0,C 180,E1 -27524.348,E2 -27524.348} C_VEL
LIN {X 0,Y 176.916,Z 689.397,A -85,B 0,C 180,E1 -27523.375,E2 -27523.375} C_VEL
LIN {X 0,Y 175.409,Z 693.201,A -85,B 0,C 180,E1 -27523.296,E2 -27523.296} C_VEL
LIN {X 0,Y 175.111,Z 693.944,A -85,B 0,C 180,E1 -27523.332,E2 -27523.332} C_VEL
LIN {X 0,Y 169.568,Z 705.989,A -85,B 0,C 180,E1 -27524.221,E2 -27524.221} C_VEL
LIN {X 0,Y 162.626,Z 717.721,A -85,B 0,C 180,E1 -27525.399,E2 -27525.399} C_VEL
LIN {X 0,Y 154.79,Z 728.524,A -85,B 0,C 180,E1 -27526.877,E2 -27526.877} C_VEL
LIN {X 0,Y 146.384,Z 737.998,A -85,B 0,C 180,E1 -27528.698,E2 -27528.698} C_VEL
LIN {X 0,Y 136.795,Z 746.933,A -85,B 0,C 180,E1 -27531.132,E2 -27531.132} C_VEL
LIN {X 0,Y 127.189,Z 754.275,A -85,B 0,C 180,E1 -27534.003,E2 -27534.003} C_VEL
LIN {X 0,Y 117.824,Z 760.165,A -85,B 0,C 180,E1 -27537.46,E2 -27537.46} C_VEL
LIN {X 0,Y 108.818,Z 764.778,A -85,B 0,C 180,E1 -27541.645,E2 -27541.645} C_VEL
LIN {X 0,Y 99.217,Z 768.532,A -85,B 0,C 180,E1 -27547.445,E2 -27547.445} C_VEL
LIN {X 0,Y 92.148,Z 770.424,A -85,B 0,C 180,E1 -27553.225,E2 -27553.225} C_VEL
LIN {X 0,Y 86.955,Z 771.203,A -85,B 0,C 180,E1 -27558.86,E2 -27558.86} C_VEL
LIN {X 0,Y 82.652,Z 771.176,A -85,B 0,C 180,E1 -27565.158,E2 -27565.158} C_VEL
LIN {X 0,Y 79.477,Z 770.382,A -85,B 0,C 180,E1 -27572.041,E2 -27572.041} C_VEL
LIN {X 0,Y 76.682,Z 767.795,A -85,B 0,C 180,E1 -27582.856,E2 -27582.856} C_VEL
LIN {X 0,Y 76.219,Z 765.221,A -85,B 0,C 180,E1 -27589.811,E2 -27589.811} C_VEL
LIN {X 0,Y 76.628,Z 761.974,A -85,B 0,C 180,E1 -27596.622,E2 -27596.622} C_VEL
LIN {X 0,Y 78.025,Z 757.247,A -85,B 0,C 180,E1 -27604.249,E2 -27604.249} C_VEL
LIN {X 0,Y 80.231,Z 751.536,A -85,B 0,C 180,E1 -27611.314,E2 -27611.314} C_VEL
LIN {X 0,Y 83.323,Z 744.654,A -85,B 0,C 180,E1 -27617.834,E2 -27617.834} C_VEL
LIN {X 0,Y 87.562,Z 735.626,A -85,B 0,C 180,E1 -27624.249,E2 -27624.249} C_VEL
LIN {X 0,Y 91.975,Z 725.755,A -85,B 0,C 180,E1 -27629.397,E2 -27629.397} C_VEL
LIN {X 0,Y 96.614,Z 714.582,A -85,B 0,C 180,E1 -27633.655,E2 -27633.655} C_VEL
LIN {X 0,Y 100.512,Z 703.859,A -85,B 0,C 180,E1 -27636.675,E2 -27636.675} C_VEL
LIN {X 0,Y 104.153,Z 691.48,A -85,B 0,C 180,E1 -27639.229,E2 -27639.229} C_VEL
LIN {X 0,Y 107.064,Z 678.949,A -85,B 0,C 180,E1 -27641.04,E2 -27641.04} C_VEL
LIN {X 0,Y 109.17,Z 666.507,A -85,B 0,C 180,E1 -27642.229,E2 -27642.229} C_VEL
LIN {X 0,Y 112.874,Z 630.152,A -85,B 0,C 180,E1 -27644.381,E2 -27644.381} C_VEL
LIN {X 0,Y 109.359,Z 621.067,A -85,B 0,C 180,E1 -27646.952,E2 -27646.952} C_VEL
LIN {X 0,Y 103.478,Z 609.316,A -85,B 0,C 180,E1 -27651.461,E2 -27651.461} C_VEL
LIN {X 0,Y 98.333,Z 600.821,A -85,B 0,C 180,E1 -27655.912,E2 -27655.912} C_VEL
LIN {X 0,Y 94.364,Z 594.572,A -85,B 0,C 180,E1 -27659.899,E2 -27659.899} C_VEL
LIN {X 0,Y 91.611,Z 590.571,A -85,B 0,C 180,E1 -27663.068,E2 -27663.068} C_VEL
LIN {X 0,Y 88.899,Z 587.134,A -85,B 0,C 180,E1 -27666.498,E2 -27666.498} C_VEL
LIN {X 0,Y 88.059,Z 585.688,A -85,B 0,C 180,E1 -27667.744,E2 -27667.744} C_VEL
LIN {X 0,Y 85.449,Z 583.202,A -85,B 0,C 180,E1 -27671.686,E2 -27671.686} C_VEL
LIN {X 0,Y 84.16,Z 580.428,A -85,B 0,C 180,E1 -27674.358,E2 -27674.358} C_VEL
LIN {X 0,Y 81.003,Z 578.294,A -85,B 0,C 180,E1 -27681.028,E2 -27681.028} C_VEL
LIN {X 0,Y 79.787,Z 575.913,A -85,B 0,C 180,E1 -27685.267,E2 -27685.267} C_VEL
LIN {X 0,Y 79.392,Z 574.586,A -85,B 0,C 180,E1 -27687.546,E2 -27687.546} C_VEL
LIN {X 0,Y 79.53,Z 574.556,A -85,B 0,C 180,E1 -27693.781,E2 -27693.781} C_VEL
LIN {X 0,Y 79.511,Z 574.565,A -85,B 0,C 180,E1 -27699.298,E2 -27699.298} C_VEL
LIN {X 0,Y 79.833,Z 574.522,A -85,B 0,C 180,E1 -27705.577,E2 -27705.577} C_VEL
LIN {X 0,Y 80.033,Z 574.489,A -85,B 0,C 180,E1 -27712.434,E2 -27712.434} C_VEL
LIN {X 0,Y 80.128,Z 574.594,A -85,B 0,C 180,E1 -27714.655,E2 -27714.655} C_VEL
LIN {X 0,Y 81.205,Z 576.867,A -85,B 0,C 180,E1 -27718.453,E2 -27718.453} C_VEL
LIN {X 0,Y 83.705,Z 579.717,A -85,B 0,C 180,E1 -27724.216,E2 -27724.216} C_VEL
LIN {X 0,Y 84.855,Z 580.542,A -85,B 0,C 180,E1 -27726.285,E2 -27726.285} C_VEL
LIN {X 0,Y 86.296,Z 583.463,A -85,B 0,C 180,E1 -27729.052,E2 -27729.052} C_VEL
LIN {X 0,Y 88.425,Z 585.746,A -85,B 0,C 180,E1 -27732.179,E2 -27732.179} C_VEL
LIN {X 0,Y 90.569,Z 589.236,A -85,B 0,C 180,E1 -27735.185,E2 -27735.185} C_VEL
LIN {X 0,Y 91.96,Z 590.939,A -85,B 0,C 180,E1 -27736.853,E2 -27736.853} C_VEL
LIN {X 0,Y 94.932,Z 595.63,A -85,B 0,C 180,E1 -27740.247,E2 -27740.247} C_VEL
LIN {X 0,Y 98.872,Z 601.825,A -85,B 0,C 180,E1 -27744.098,E2 -27744.098} C_VEL
LIN {X 0,Y 104.721,Z 612.645,A -85,B 0,C 180,E1 -27749.177,E2 -27749.177} C_VEL
LIN {X 0,Y 107.118,Z 618.546,A -85,B 0,C 180,E1 -27751.154,E2 -27751.154} C_VEL
LIN {X 0,Y 111.091,Z 630.733,A -85,B 0,C 180,E1 -27754.39,E2 -27754.39} C_VEL
LIN {X 0,Y 112.639,Z 636.207,A -85,B 0,C 180,E1 -27755.644,E2 -27755.644} C_VEL
LIN {X 0,Y 108.772,Z 673.224,A -85,B 0,C 180,E1 -27757.878,E2 -27757.878} C_VEL
LIN {X 0,Y 106.187,Z 687.266,A -85,B 0,C 180,E1 -27759.319,E2 -27759.319} C_VEL
LIN {X 0,Y 102.889,Z 699.85,A -85,B 0,C 180,E1 -27761.283,E2 -27761.283} C_VEL
LIN {X 0,Y 98.939,Z 712.006,A -85,B 0,C 180,E1 -27764.002,E2 -27764.002} C_VEL
LIN {X 0,Y 94.76,Z 723.014,A -85,B 0,C 180,E1 -27767.401,E2 -27767.401} C_VEL
LIN {X 0,Y 90.446,Z 732.95,A -85,B 0,C 180,E1 -27771.557,E2 -27771.557} C_VEL
LIN {X 0,Y 86.266,Z 741.982,A -85,B 0,C 180,E1 -27776.631,E2 -27776.631} C_VEL
LIN {X 0,Y 82.193,Z 750.802,A -85,B 0,C 180,E1 -27783.319,E2 -27783.319} C_VEL
LIN {X 0,Y 79.243,Z 757.809,A -85,B 0,C 180,E1 -27790.567,E2 -27790.567} C_VEL
LIN {X 0,Y 77.79,Z 762.583,A -85,B 0,C 180,E1 -27796.939,E2 -27796.939} C_VEL
LIN {X 0,Y 77.019,Z 767.111,A -85,B 0,C 180,E1 -27804.757,E2 -27804.757} C_VEL
LIN {X 0,Y 77.028,Z 769.458,A -85,B 0,C 180,E1 -27809.993,E2 -27809.993} C_VEL
LIN {X 0,Y 76.962,Z 771.308,A -85,B 0,C 180,E1 -27815.232,E2 -27815.232} C_VEL
LIN {X 0,Y 77.316,Z 772.747,A -85,B 0,C 180,E1 -27820.467,E2 -27820.467} C_VEL
LIN {X 0,Y 78.175,Z 773.795,A -85,B 0,C 180,E1 -27825.639,E2 -27825.639} C_VEL
LIN {X 0,Y 81.67,Z 774.72,A -85,B 0,C 180,E1 -27835.476,E2 -27835.476} C_VEL
LIN {X 0,Y 87.579,Z 774.23,A -85,B 0,C 180,E1 -27844.167,E2 -27844.167} C_VEL
LIN {X 0,Y 95.282,Z 772.286,A -85,B 0,C 180,E1 -27851.585,E2 -27851.585} C_VEL
LIN {X 0,Y 104.33,Z 768.812,A -85,B 0,C 180,E1 -27857.807,E2 -27857.807} C_VEL
LIN {X 0,Y 111.893,Z 765.149,A -85,B 0,C 180,E1 -27861.724,E2 -27861.724} C_VEL
LIN {X 0,Y 120.058,Z 760.451,A -85,B 0,C 180,E1 -27865.029,E2 -27865.029} C_VEL
LIN {X 0,Y 128.536,Z 754.637,A -85,B 0,C 180,E1 -27867.931,E2 -27867.931} C_VEL
LIN {X 0,Y 137.386,Z 747.508,A -85,B 0,C 180,E1 -27870.407,E2 -27870.407} C_VEL
LIN {X 0,Y 146.512,Z 738.765,A -85,B 0,C 180,E1 -27872.541,E2 -27872.541} C_VEL
LIN {X 0,Y 154.32,Z 729.843,A -85,B 0,C 180,E1 -27874.076,E2 -27874.076} C_VEL
LIN {X 0,Y 162.253,Z 718.853,A -85,B 0,C 180,E1 -27875.443,E2 -27875.443} C_VEL
LIN {X 0,Y 168.715,Z 708.013,A -85,B 0,C 180,E1 -27876.4,E2 -27876.4} C_VEL
LIN {X 0,Y 173.956,Z 697.113,A -85,B 0,C 180,E1 -27877.117,E2 -27877.117} C_VEL
LIN {X 0,Y 178.436,Z 685.152,A -85,B 0,C 180,E1 -27877.638,E2 -27877.638} C_VEL
LIN {X 0,Y 179.607,Z 681.295,A -85,B 0,C 180,E1 -27877.78,E2 -27877.78} C_VEL
LIN {X 0,Y 179.757,Z 680.044,A -85,B 0,C 180,E1 -27879.397,E2 -27879.397} C_VEL
LIN {X 0,Y 179.852,Z 679.807,A -85,B 0,C 180,E1 -27881.782,E2 -27881.782} C_VEL
LIN {X 0,Y 179.902,Z 680.004,A -85,B 0,C 180,E1 -27882.61,E2 -27882.61} C_VEL
LIN {X 0,Y 175.563,Z 692.801,A -85,B 0,C 180,E1 -27883.261,E2 -27883.261} C_VEL
LIN {X 0,Y 175.111,Z 693.944,A -85,B 0,C 180,E1 -27883.332,E2 -27883.332} C_VEL
LIN {X 0,Y 172.772,Z 699.361,A -85,B 0,C 180,E1 -27883.473,E2 -27883.473} C_VEL
LIN {X 0,Y 168.213,Z 708.134,A -85,B 0,C 180,E1 -27883.19,E2 -27883.19} C_VEL
LIN {X 0,Y 163.027,Z 716.511,A -85,B 0,C 180,E1 -27882.969,E2 -27882.969} C_VEL
LIN {X 0,Y 159.701,Z 721.299,A -85,B 0,C 180,E1 -27883.239,E2 -27883.239} C_VEL
LIN {X 0,Y 152.219,Z 730.766,A -85,B 0,C 180,E1 -27884.521,E2 -27884.521} C_VEL
LIN {X 0,Y 144.834,Z 738.632,A -85,B 0,C 180,E1 -27885.957,E2 -27885.957} C_VEL
LIN {X 0,Y 134.841,Z 747.566,A -85,B 0,C 180,E1 -27888.217,E2 -27888.217} C_VEL
LIN {X 0,Y 126.564,Z 753.699,A -85,B 0,C 180,E1 -27890.409,E2 -27890.409} C_VEL
LIN {X 0,Y 117.873,Z 759.109,A -85,B 0,C 180,E1 -27893.15,E2 -27893.15} C_VEL
LIN {X 0,Y 109.624,Z 763.361,A -85,B 0,C 180,E1 -27896.322,E2 -27896.322} C_VEL
LIN {X 0,Y 101.801,Z 766.655,A -85,B 0,C 180,E1 -27899.998,E2 -27899.998} C_VEL
LIN {X 0,Y 91.877,Z 769.792,A -85,B 0,C 180,E1 -27906.12,E2 -27906.12} C_VEL
LIN {X 0,Y 85.91,Z 770.981,A -85,B 0,C 180,E1 -27911.021,E2 -27911.021} C_VEL
LIN {X 0,Y 80.665,Z 771.488,A -85,B 0,C 180,E1 -27916.613,E2 -27916.613} C_VEL
LIN {X 0,Y 76.279,Z 771.334,A -85,B 0,C 180,E1 -27922.895,E2 -27922.895} C_VEL
LIN {X 0,Y 72.939,Z 770.434,A -85,B 0,C 180,E1 -27929.883,E2 -27929.883} C_VEL
LIN {X 0,Y 69.834,Z 767.871,A -85,B 0,C 180,E1 -27941.006,E2 -27941.006} C_VEL
LIN {X 0,Y 69.165,Z 765.193,A -85,B 0,C 180,E1 -27948.872,E2 -27948.872} C_VEL
LIN {X 0,Y 69.568,Z 761.542,A -85,B 0,C 180,E1 -27957.073,E2 -27957.073} C_VEL
LIN {X 0,Y 71.045,Z 756.824,A -85,B 0,C 180,E1 -27965.185,E2 -27965.185} C_VEL
LIN {X 0,Y 73.652,Z 750.542,A -85,B 0,C 180,E1 -27973.374,E2 -27973.374} C_VEL
LIN {X 0,Y 77.413,Z 742.753,A -85,B 0,C 180,E1 -27980.91,E2 -27980.91} C_VEL
LIN {X 0,Y 82.136,Z 733.217,A -85,B 0,C 180,E1 -27987.555,E2 -27987.555} C_VEL
LIN {X 0,Y 87.116,Z 722.613,A -85,B 0,C 180,E1 -27992.897,E2 -27992.897} C_VEL
LIN {X 0,Y 92.06,Z 710.878,A -85,B 0,C 180,E1 -27997.067,E2 -27997.067} C_VEL
LIN {X 0,Y 96.379,Z 698.565,A -85,B 0,C 180,E1 -28000.244,E2 -28000.244} C_VEL
LIN {X 0,Y 100.036,Z 685.664,A -85,B 0,C 180,E1 -28002.529,E2 -28002.529} C_VEL
LIN {X 0,Y 102.79,Z 672.051,A -85,B 0,C 180,E1 -28004.21,E2 -28004.21} C_VEL
LIN {X 0,Y 104.73,Z 657.588,A -85,B 0,C 180,E1 -28005.222,E2 -28005.222} C_VEL
LIN {X 0,Y 107.407,Z 632.49,A -85,B 0,C 180,E1 -28006.665,E2 -28006.665} C_VEL
LIN {X 0,Y 104.745,Z 625.126,A -85,B 0,C 180,E1 -28008.853,E2 -28008.853} C_VEL
LIN {X 0,Y 99.368,Z 613.953,A -85,B 0,C 180,E1 -28013.457,E2 -28013.457} C_VEL
LIN {X 0,Y 94.617,Z 605.787,A -85,B 0,C 180,E1 -28017.978,E2 -28017.978} C_VEL
LIN {X 0,Y 91.096,Z 600.057,A -85,B 0,C 180,E1 -28021.94,E2 -28021.94} C_VEL
LIN {X 0,Y 88.155,Z 595.796,A -85,B 0,C 180,E1 -28025.652,E2 -28025.652} C_VEL
LIN {X 0,Y 85.583,Z 591.972,A -85,B 0,C 180,E1 -28029.487,E2 -28029.487} C_VEL
LIN {X 0,Y 83.163,Z 589.251,A -85,B 0,C 180,E1 -28033.651,E2 -28033.651} C_VEL
LIN {X 0,Y 82.126,Z 587.078,A -85,B 0,C 180,E1 -28035.952,E2 -28035.952} C_VEL
LIN {X 0,Y 79.127,Z 584.566,A -85,B 0,C 180,E1 -28043.291,E2 -28043.291} C_VEL
LIN {X 0,Y 77.942,Z 581.507,A -85,B 0,C 180,E1 -28048.773,E2 -28048.773} C_VEL
LIN {X 0,Y 76.91,Z 581.066,A -85,B 0,C 180,E1 -28064.092,E2 -28064.092} C_VEL
LIN {X 0,Y 78.709,Z 581.635,A -85,B 0,C 180,E1 -28073.593,E2 -28073.593} C_VEL
LIN {X 0,Y 81.816,Z 586.318,A -85,B 0,C 180,E1 -28082.772,E2 -28082.772} C_VEL
LIN {X 0,Y 82.719,Z 587.097,A -85,B 0,C 180,E1 -28084.571,E2 -28084.571} C_VEL
LIN {X 0,Y 84.576,Z 590.448,A -85,B 0,C 180,E1 -28088.298,E2 -28088.298} C_VEL
LIN {X 0,Y 85.959,Z 592.076,A -85,B 0,C 180,E1 -28090.519,E2 -28090.519} C_VEL
LIN {X 0,Y 88.529,Z 596.002,A -85,B 0,C 180,E1 -28094.275,E2 -28094.275} C_VEL
LIN {X 0,Y 91.588,Z 600.934,A -85,B 0,C 180,E1 -28098.189,E2 -28098.189} C_VEL
LIN {X 0,Y 95.51,Z 607.553,A -85,B 0,C 180,E1 -28102.48,E2 -28102.48} C_VEL
LIN {X 0,Y 100.711,Z 617.6,A -85,B 0,C 180,E1 -28107.398,E2 -28107.398} C_VEL
LIN {X 0,Y 103.953,Z 626.752,A -85,B 0,C 180,E1 -28110.411,E2 -28110.411} C_VEL
LIN {X 0,Y 107.135,Z 637.855,A -85,B 0,C 180,E1 -28113.288,E2 -28113.288} C_VEL
LIN {X 0,Y 103.286,Z 673.08,A -85,B 0,C 180,E1 -28115.463,E2 -28115.463} C_VEL
LIN {X 0,Y 100.571,Z 687.148,A -85,B 0,C 180,E1 -28116.932,E2 -28116.932} C_VEL
LIN {X 0,Y 97.132,Z 699.675,A -85,B 0,C 180,E1 -28118.93,E2 -28118.93} C_VEL
LIN {X 0,Y 92.983,Z 711.789,A -85,B 0,C 180,E1 -28121.713,E2 -28121.713} C_VEL
LIN {X 0,Y 88.53,Z 722.885,A -85,B 0,C 180,E1 -28125.272,E2 -28125.272} C_VEL
LIN {X 0,Y 84.022,Z 732.697,A -85,B 0,C 180,E1 -28129.582,E2 -28129.582} C_VEL
LIN {X 0,Y 79.598,Z 741.738,A -85,B 0,C 180,E1 -28134.968,E2 -28134.968} C_VEL
LIN {X 0,Y 75.93,Z 749.205,A -85,B 0,C 180,E1 -28140.918,E2 -28140.918} C_VEL
LIN {X 0,Y 72.569,Z 756.511,A -85,B 0,C 180,E1 -28148.697,E2 -28148.697} C_VEL
LIN {X 0,Y 70.883,Z 761.446,A -85,B 0,C 180,E1 -28155.64,E2 -28155.64} C_VEL
LIN {X 0,Y 69.992,Z 766.185,A -85,B 0,C 180,E1 -28164.229,E2 -28164.229} C_VEL
LIN {X 0,Y 69.95,Z 768.696,A -85,B 0,C 180,E1 -28169.992,E2 -28169.992} C_VEL
LIN {X 0,Y 69.918,Z 770.633,A -85,B 0,C 180,E1 -28175.761,E2 -28175.761} C_VEL
LIN {X 0,Y 71.355,Z 773.28,A -85,B 0,C 180,E1 -28187.178,E2 -28187.178} C_VEL
LIN {X 0,Y 75.3,Z 774.461,A -85,B 0,C 180,E1 -28197.809,E2 -28197.809} C_VEL
LIN {X 0,Y 81.789,Z 774.159,A -85,B 0,C 180,E1 -28206.968,E2 -28206.968} C_VEL
LIN {X 0,Y 90.101,Z 772.44,A -85,B 0,C 180,E1 -28214.579,E2 -28214.579} C_VEL
LIN {X 0,Y 99.711,Z 769.239,A -85,B 0,C 180,E1 -28220.824,E2 -28220.824} C_VEL
LIN {X 0,Y 107.663,Z 765.781,A -85,B 0,C 180,E1 -28224.673,E2 -28224.673} C_VEL
LIN {X 0,Y 116.173,Z 761.333,A -85,B 0,C 180,E1 -28227.871,E2 -28227.871} C_VEL
LIN {X 0,Y 124.958,Z 755.805,A -85,B 0,C 180,E1 -28230.654,E2 -28230.654} C_VEL
LIN {X 0,Y 134.088,Z 748.983,A -85,B 0,C 180,E1 -28232.992,E2 -28232.992} C_VEL
LIN {X 0,Y 143.441,Z 740.586,A -85,B 0,C 180,E1 -28235.005,E2 -28235.005} C_VEL
LIN {X 0,Y 151.416,Z 732.14,A -85,B 0,C 180,E1 -28236.437,E2 -28236.437} C_VEL
LIN {X 0,Y 159.511,Z 721.878,A -85,B 0,C 180,E1 -28237.696,E2 -28237.696} C_VEL
LIN {X 0,Y 166.102,Z 711.761,A -85,B 0,C 180,E1 -28238.557,E2 -28238.557} C_VEL
LIN {X 0,Y 171.882,Z 700.844,A -85,B 0,C 180,E1 -28239.27,E2 -28239.27} C_VEL
LIN {X 0,Y 176.987,Z 688.444,A -85,B 0,C 180,E1 -28239.808,E2 -28239.808} C_VEL
LIN {X 0,Y 177.6,Z 686.669,A -85,B 0,C 180,E1 -28240.114,E2 -28240.114} C_VEL
LIN {X 0,Y 177.593,Z 686.639,A -85,B 0,C 180,E1 -28240.439,E2 -28240.439} C_VEL
LIN {X 0,Y 177.167,Z 687.853,A -85,B 0,C 180,E1 -28240.667,E2 -28240.667} C_VEL
LIN {X 0,Y 172.043,Z 700.355,A -85,B 0,C 180,E1 -28241.378,E2 -28241.378} C_VEL
LIN {X 0,Y 165.728,Z 712.143,A -85,B 0,C 180,E1 -28242.298,E2 -28242.298} C_VEL
LIN {X 0,Y 159.701,Z 721.299,A -85,B 0,C 180,E1 -28243.239,E2 -28243.239} C_VEL
LIN {X 0,Y 156.127,Z 726.011,A -85,B 0,C 180,E1 -28243.556,E2 -28243.556} C_VEL
LIN {X 0,Y 149.564,Z 733.543,A -85,B 0,C 180,E1 -28243.526,E2 -28243.526} C_VEL
LIN {X 0,Y 142.56,Z 740.42,A -85,B 0,C 180,E1 -28243.624,E2 -28243.624} C_VEL
LIN {X 0,Y 138.328,Z 744.149,A -85,B 0,C 180,E1 -28244.186,E2 -28244.186} C_VEL
LIN {X 0,Y 129.005,Z 751.382,A -85,B 0,C 180,E1 -28246.2,E2 -28246.2} C_VEL
LIN {X 0,Y 118.941,Z 757.776,A -85,B 0,C 180,E1 -28248.784,E2 -28248.784} C_VEL
LIN {X 0,Y 110.558,Z 762.204,A -85,B 0,C 180,E1 -28251.424,E2 -28251.424} C_VEL
LIN {X 0,Y 99.292,Z 766.856,A -85,B 0,C 180,E1 -28255.939,E2 -28255.939} C_VEL
LIN {X 0,Y 91.353,Z 769.295,A -85,B 0,C 180,E1 -28260.078,E2 -28260.078} C_VEL
LIN {X 0,Y 84.308,Z 770.855,A -85,B 0,C 180,E1 -28264.779,E2 -28264.779} C_VEL
LIN {X 0,Y 77.833,Z 771.644,A -85,B 0,C 180,E1 -28270.401,E2 -28270.401} C_VEL
LIN {X 0,Y 72.193,Z 771.65,A -85,B 0,C 180,E1 -28276.978,E2 -28276.978} C_VEL
LIN {X 0,Y 67.707,Z 770.899,A -85,B 0,C 180,E1 -28284.528,E2 -28284.528} C_VEL
LIN {X 0,Y 64.423,Z 769.357,A -85,B 0,C 180,E1 -28293.052,E2 -28293.052} C_VEL
LIN {X 0,Y 62.497,Z 766.883,A -85,B 0,C 180,E1 -28302.428,E2 -28302.428} C_VEL
LIN {X 0,Y 62.104,Z 763.357,A -85,B 0,C 180,E1 -28312.382,E2 -28312.382} C_VEL
LIN {X 0,Y 63.544,Z 757.86,A -85,B 0,C 180,E1 -28323.753,E2 -28323.753} C_VEL
LIN {X 0,Y 66.121,Z 751.693,A -85,B 0,C 180,E1 -28333.05,E2 -28333.05} C_VEL
LIN {X 0,Y 70.318,Z 743.456,A -85,B 0,C 180,E1 -28342.06,E2 -28342.06} C_VEL
LIN {X 0,Y 74.84,Z 734.979,A -85,B 0,C 180,E1 -28348.662,E2 -28348.662} C_VEL
LIN {X 0,Y 80.049,Z 724.589,A -85,B 0,C 180,E1 -28354.466,E2 -28354.466} C_VEL
LIN {X 0,Y 85.104,Z 713.545,A -85,B 0,C 180,E1 -28358.844,E2 -28358.844} C_VEL
LIN {X 0,Y 89.328,Z 702.739,A -85,B 0,C 180,E1 -28361.925,E2 -28361.925} C_VEL
LIN {X 0,Y 93.228,Z 690.511,A -85,B 0,C 180,E1 -28364.459,E2 -28364.459} C_VEL
LIN {X 0,Y 96.34,Z 677.957,A -85,B 0,C 180,E1 -28366.265,E2 -28366.265} C_VEL
LIN {X 0,Y 98.68,Z 664.564,A -85,B 0,C 180,E1 -28367.444,E2 -28367.444} C_VEL
LIN {X 0,Y 101.981,Z 634.067,A -85,B 0,C 180,E1 -28369.322,E2 -28369.322} C_VEL
LIN {X 0,Y 100.177,Z 629.058,A -85,B 0,C 180,E1 -28370.994,E2 -28370.994} C_VEL
LIN {X 0,Y 95.1,Z 618.064,A -85,B 0,C 180,E1 -28375.807,E2 -28375.807} C_VEL
LIN {X 0,Y 89.819,Z 608.533,A -85,B 0,C 180,E1 -28381.7,E2 -28381.7} C_VEL
LIN {X 0,Y 87.062,Z 604.297,A -85,B 0,C 180,E1 -28385.217,E2 -28385.217} C_VEL
LIN {X 0,Y 85.324,Z 601.547,A -85,B 0,C 180,E1 -28387.754,E2 -28387.754} C_VEL
LIN {X 0,Y 83.06,Z 598.104,A -85,B 0,C 180,E1 -28391.56,E2 -28391.56} C_VEL
LIN {X 0,Y 80.716,Z 594.904,A -85,B 0,C 180,E1 -28396.195,E2 -28396.195} C_VEL
LIN {X 0,Y 80.145,Z 593.714,A -85,B 0,C 180,E1 -28397.618,E2 -28397.618} C_VEL
LIN {X 0,Y 77.448,Z 590.922,A -85,B 0,C 180,E1 -28405.341,E2 -28405.341} C_VEL
LIN {X 0,Y 76.649,Z 588.484,A -85,B 0,C 180,E1 -28409.718,E2 -28409.718} C_VEL
LIN {X 0,Y 75.823,Z 588.087,A -85,B 0,C 180,E1 -28423.858,E2 -28423.858} C_VEL
LIN {X 0,Y 77.336,Z 588.602,A -85,B 0,C 180,E1 -28432.569,E2 -28432.569} C_VEL
LIN {X 0,Y 80.24,Z 593.129,A -85,B 0,C 180,E1 -28441.885,E2 -28441.885} C_VEL
LIN {X 0,Y 80.85,Z 593.991,A -85,B 0,C 180,E1 -28443.273,E2 -28443.273} C_VEL
LIN {X 0,Y 82.851,Z 597.284,A -85,B 0,C 180,E1 -28447.444,E2 -28447.444} C_VEL
LIN {X 0,Y 83.99,Z 599.21,A -85,B 0,C 180,E1 -28449.53,E2 -28449.53} C_VEL
LIN {X 0,Y 86.954,Z 603.818,A -85,B 0,C 180,E1 -28454.071,E2 -28454.071} C_VEL
LIN {X 0,Y 91.351,Z 611.558,A -85,B 0,C 180,E1 -28459.725,E2 -28459.725} C_VEL
LIN {X 0,Y 96.285,Z 621.458,A -85,B 0,C 180,E1 -28465.001,E2 -28465.001} C_VEL
LIN {X 0,Y 98.516,Z 627.635,A -85,B 0,C 180,E1 -28467.305,E2 -28467.305} C_VEL
LIN {X 0,Y 101.605,Z 638.713,A -85,B 0,C 180,E1 -28470.53,E2 -28470.53} C_VEL
LIN {X 0,Y 101.706,Z 640.419,A -85,B 0,C 180,E1 -28470.79,E2 -28470.79} C_VEL
LIN {X 0,Y 97.881,Z 673.329,A -85,B 0,C 180,E1 -28472.845,E2 -28472.845} C_VEL
LIN {X 0,Y 95.142,Z 686.804,A -85,B 0,C 180,E1 -28474.259,E2 -28474.259} C_VEL
LIN {X 0,Y 91.552,Z 699.382,A -85,B 0,C 180,E1 -28476.28,E2 -28476.28} C_VEL
LIN {X 0,Y 87.191,Z 711.508,A -85,B 0,C 180,E1 -28479.111,E2 -28479.111} C_VEL
LIN {X 0,Y 82.212,Z 723.218,A -85,B 0,C 180,E1 -28483.022,E2 -28483.022} C_VEL
LIN {X 0,Y 76.691,Z 734.393,A -85,B 0,C 180,E1 -28488.355,E2 -28488.355} C_VEL
LIN {X 0,Y 72.173,Z 743.138,A -85,B 0,C 180,E1 -28494.24,E2 -28494.24} C_VEL
LIN {X 0,Y 67.736,Z 751.581,A -85,B 0,C 180,E1 -28502.157,E2 -28502.157} C_VEL
LIN {X 0,Y 64.698,Z 758.338,A -85,B 0,C 180,E1 -28510.972,E2 -28510.972} C_VEL
LIN {X 0,Y 63.147,Z 763.7,A -85,B 0,C 180,E1 -28520.381,E2 -28520.381} C_VEL
LIN {X 0,Y 62.89,Z 767.814,A -85,B 0,C 180,E1 -28529.991,E2 -28529.991} C_VEL
LIN {X 0,Y 62.894,Z 769.901,A -85,B 0,C 180,E1 -28536.407,E2 -28536.407} C_VEL
LIN {X 0,Y 63.418,Z 771.535,A -85,B 0,C 180,E1 -28542.796,E2 -28542.796} C_VEL
LIN {X 0,Y 66.517,Z 773.62,A -85,B 0,C 180,E1 -28554.991,E2 -28554.991} C_VEL
LIN {X 0,Y 72.392,Z 774.282,A -85,B 0,C 180,E1 -28565.616,E2 -28565.616} C_VEL
LIN {X 0,Y 80.484,Z 773.51,A -85,B 0,C 180,E1 -28574.302,E2 -28574.302} C_VEL
LIN {X 0,Y 90.154,Z 771.271,A -85,B 0,C 180,E1 -28581.209,E2 -28581.209} C_VEL
LIN {X 0,Y 100.888,Z 767.58,A -85,B 0,C 180,E1 -28586.702,E2 -28586.702} C_VEL
LIN {X 0,Y 109.613,Z 763.681,A -85,B 0,C 180,E1 -28589.936,E2 -28589.936} C_VEL
LIN {X 0,Y 118.573,Z 758.779,A -85,B 0,C 180,E1 -28592.746,E2 -28592.746} C_VEL
LIN {X 0,Y 129.488,Z 751.574,A -85,B 0,C 180,E1 -28595.371,E2 -28595.371} C_VEL
LIN {X 0,Y 139.035,Z 743.889,A -85,B 0,C 180,E1 -28597.284,E2 -28597.284} C_VEL
LIN {X 0,Y 148.791,Z 734.421,A -85,B 0,C 180,E1 -28598.875,E2 -28598.875} C_VEL
LIN {X 0,Y 157.034,Z 724.707,A -85,B 0,C 180,E1 -28600.014,E2 -28600.014} C_VEL
LIN {X 0,Y 158.291,Z 722.97,A -85,B 0,C 180,E1 -28600.802,E2 -28600.802} C_VEL
LIN {X 0,Y 150.576,Z 732.298,A -85,B 0,C 180,E1 -28601.973,E2 -28601.973} C_VEL
LIN {X 0,Y 142.632,Z 740.328,A -85,B 0,C 180,E1 -28603.347,E2 -28603.347} C_VEL
LIN {X 0,Y 138.328,Z 744.149,A -85,B 0,C 180,E1 -28604.186,E2 -28604.186} C_VEL
LIN {X 0,Y 133.888,Z 747.757,A -85,B 0,C 180,E1 -28604.824,E2 -28604.824} C_VEL
LIN {X 0,Y 125.759,Z 753.397,A -85,B 0,C 180,E1 -28605.222,E2 -28605.222} C_VEL
LIN {X 0,Y 117.279,Z 758.394,A -85,B 0,C 180,E1 -28605.749,E2 -28605.749} C_VEL
LIN {X 0,Y 112.329,Z 760.899,A -85,B 0,C 180,E1 -28606.685,E2 -28606.685} C_VEL
LIN {X 0,Y 102.872,Z 765.056,A -85,B 0,C 180,E1 -28609.645,E2 -28609.645} C_VEL
LIN {X 0,Y 91.847,Z 768.743,A -85,B 0,C 180,E1 -28614.057,E2 -28614.057} C_VEL
LIN {X 0,Y 81.191,Z 771.084,A -85,B 0,C 180,E1 -28619.997,E2 -28619.997} C_VEL
LIN {X 0,Y 71.011,Z 771.967,A -85,B 0,C 180,E1 -28628.29,E2 -28628.29} C_VEL
LIN {X 0,Y 65.434,Z 771.694,A -85,B 0,C 180,E1 -28634.875,E2 -28634.875} C_VEL
LIN {X 0,Y 60.898,Z 770.728,A -85,B 0,C 180,E1 -28642.62,E2 -28642.62} C_VEL
LIN {X 0,Y 57.573,Z 769.058,A -85,B 0,C 180,E1 -28651.316,E2 -28651.316} C_VEL
LIN {X 0,Y 55.602,Z 766.731,A -85,B 0,C 180,E1 -28660.694,E2 -28660.694} C_VEL
LIN {X 0,Y 54.98,Z 763.69,A -85,B 0,C 180,E1 -28670.286,E2 -28670.286} C_VEL
LIN {X 0,Y 55.932,Z 759.026,A -85,B 0,C 180,E1 -28681.582,E2 -28681.582} C_VEL
LIN {X 0,Y 58.737,Z 752.442,A -85,B 0,C 180,E1 -28693.165,E2 -28693.165} C_VEL
LIN {X 0,Y 62.463,Z 745.513,A -85,B 0,C 180,E1 -28701.924,E2 -28701.924} C_VEL
LIN {X 0,Y 67.51,Z 736.556,A -85,B 0,C 180,E1 -28710.009,E2 -28710.009} C_VEL
LIN {X 0,Y 72.978,Z 726.596,A -85,B 0,C 180,E1 -28716.228,E2 -28716.228} C_VEL
LIN {X 0,Y 78.488,Z 715.481,A -85,B 0,C 180,E1 -28721.047,E2 -28721.047} C_VEL
LIN {X 0,Y 83.475,Z 703.714,A -85,B 0,C 180,E1 -28724.637,E2 -28724.637} C_VEL
LIN {X 0,Y 87.588,Z 691.617,A -85,B 0,C 180,E1 -28727.238,E2 -28727.238} C_VEL
LIN {X 0,Y 91.027,Z 678.666,A -85,B 0,C 180,E1 -28729.145,E2 -28729.145} C_VEL
LIN {X 0,Y 93.437,Z 665.686,A -85,B 0,C 180,E1 -28730.341,E2 -28730.341} C_VEL
LIN {X 0,Y 96.923,Z 636.13,A -85,B 0,C 180,E1 -28732.117,E2 -28732.117} C_VEL
LIN {X 0,Y 94.705,Z 630.708,A -85,B 0,C 180,E1 -28734.305,E2 -28734.305} C_VEL
LIN {X 0,Y 91.346,Z 622.977,A -85,B 0,C 180,E1 -28737.969,E2 -28737.969} C_VEL
LIN {X 0,Y 86.472,Z 613.663,A -85,B 0,C 180,E1 -28744.067,E2 -28744.067} C_VEL
LIN {X 0,Y 82.796,Z 607.57,A -85,B 0,C 180,E1 -28749.684,E2 -28749.684} C_VEL
LIN {X 0,Y 80.868,Z 604.439,A -85,B 0,C 180,E1 -28753.328,E2 -28753.328} C_VEL
LIN {X 0,Y 78.489,Z 600.696,A -85,B 0,C 180,E1 -28758.694,E2 -28758.694} C_VEL
LIN {X 0,Y 75.723,Z 596.943,A -85,B 0,C 180,E1 -28768.142,E2 -28768.142} C_VEL
LIN {X 0,Y 75.379,Z 595.446,A -85,B 0,C 180,E1 -28770.696,E2 -28770.696} C_VEL
LIN {X 0,Y 74.737,Z 595.108,A -85,B 0,C 180,E1 -28783.617,E2 -28783.617} C_VEL
LIN {X 0,Y 75.979,Z 595.497,A -85,B 0,C 180,E1 -28791.444,E2 -28791.444} C_VEL
LIN {X 0,Y 78.788,Z 600.251,A -85,B 0,C 180,E1 -28801.28,E2 -28801.28} C_VEL
LIN {X 0,Y 81.367,Z 604.758,A -85,B 0,C 180,E1 -28807.073,E2 -28807.073} C_VEL
LIN {X 0,Y 84.583,Z 610.306,A -85,B 0,C 180,E1 -28812.682,E2 -28812.682} C_VEL
LIN {X 0,Y 88.619,Z 618.01,A -85,B 0,C 180,E1 -28818.329,E2 -28818.329} C_VEL
LIN {X 0,Y 92.891,Z 627.483,A -85,B 0,C 180,E1 -28823.427,E2 -28823.427} C_VEL
LIN {X 0,Y 96.24,Z 639.207,A -85,B 0,C 180,E1 -28827.36,E2 -28827.36} C_VEL
LIN {X 0,Y 96.617,Z 640.882,A -85,B 0,C 180,E1 -28827.828,E2 -28827.828} C_VEL
LIN {X 0,Y 92.784,Z 673.099,A -85,B 0,C 180,E1 -28829.888,E2 -28829.888} C_VEL
LIN {X 0,Y 89.948,Z 686.465,A -85,B 0,C 180,E1 -28831.274,E2 -28831.274} C_VEL
LIN {X 0,Y 86.192,Z 699.058,A -85,B 0,C 180,E1 -28833.292,E2 -28833.292} C_VEL
LIN {X 0,Y 81.611,Z 711.175,A -85,B 0,C 180,E1 -28836.152,E2 -28836.152} C_VEL
LIN {X 0,Y 76.538,Z 722.51,A -85,B 0,C 180,E1 -28840.002,E2 -28840.002} C_VEL
LIN {X 0,Y 71.556,Z 732.108,A -85,B 0,C 180,E1 -28844.586,E2 -28844.586} C_VEL
LIN {X 0,Y 66.531,Z 741.157,A -85,B 0,C 180,E1 -28850.657,E2 -28850.657} C_VEL
LIN {X 0,Y 61.541,Z 749.974,A -85,B 0,C 180,E1 -28859.065,E2 -28859.065} C_VEL
LIN {X 0,Y 58.019,Z 757.005,A -85,B 0,C 180,E1 -28868.68,E2 -28868.68} C_VEL
LIN {X 0,Y 56.187,Z 762.597,A -85,B 0,C 180,E1 -28879.176,E2 -28879.176} C_VEL
LIN {X 0,Y 55.845,Z 766.922,A -85,B 0,C 180,E1 -28889.99,E2 -28889.99} C_VEL
LIN {X 0,Y 55.887,Z 769.105,A -85,B 0,C 180,E1 -28897.214,E2 -28897.214} C_VEL
LIN {X 0,Y 56.537,Z 770.853,A -85,B 0,C 180,E1 -28904.385,E2 -28904.385} C_VEL
LIN {X 0,Y 60.152,Z 773.173,A -85,B 0,C 180,E1 -28917.851,E2 -28917.851} C_VEL
LIN {X 0,Y 66.734,Z 774.027,A -85,B 0,C 180,E1 -28929.178,E2 -28929.178} C_VEL
LIN {X 0,Y 75.564,Z 773.491,A -85,B 0,C 180,E1 -28938.067,E2 -28938.067} C_VEL
LIN {X 0,Y 85.883,Z 771.53,A -85,B 0,C 180,E1 -28944.905,E2 -28944.905} C_VEL
LIN {X 0,Y 97.181,Z 768.056,A -85,B 0,C 180,E1 -28950.194,E2 -28950.194} C_VEL
LIN {X 0,Y 106.256,Z 764.39,A -85,B 0,C 180,E1 -28953.229,E2 -28953.229} C_VEL
LIN {X 0,Y 115.527,Z 759.775,A -85,B 0,C 180,E1 -28955.842,E2 -28955.842} C_VEL
LIN {X 0,Y 126.742,Z 752.916,A -85,B 0,C 180,E1 -28958.237,E2 -28958.237} C_VEL
LIN {X 0,Y 136.681,Z 745.465,A -85,B 0,C 180,E1 -28959.996,E2 -28959.996} C_VEL
LIN {X 0,Y 138.154,Z 744.216,A -85,B 0,C 180,E1 -28960.225,E2 -28960.225} C_VEL
LIN {X 0,Y 139.336,Z 743.161,A -85,B 0,C 180,E1 -28960.891,E2 -28960.891} C_VEL
LIN {X 0,Y 128.692,Z 751.364,A -85,B 0,C 180,E1 -28962.858,E2 -28962.858} C_VEL
LIN {X 0,Y 118.129,Z 757.898,A -85,B 0,C 180,E1 -28965.169,E2 -28965.169} C_VEL
LIN {X 0,Y 112.329,Z 760.899,A -85,B 0,C 180,E1 -28966.685,E2 -28966.685} C_VEL
LIN {X 0,Y 107.286,Z 763.231,A -85,B 0,C 180,E1 -28967.759,E2 -28967.759} C_VEL
LIN {X 0,Y 98.185,Z 766.646,A -85,B 0,C 180,E1 -28968.898,E2 -28968.898} C_VEL
LIN {X 0,Y 88.971,Z 769.298,A -85,B 0,C 180,E1 -28970.381,E2 -28970.381} C_VEL
LIN {X 0,Y 83.844,Z 770.372,A -85,B 0,C 180,E1 -28972.155,E2 -28972.155} C_VEL
LIN {X 0,Y 77.533,Z 771.46,A -85,B 0,C 180,E1 -28975.531,E2 -28975.531} C_VEL
LIN {X 0,Y 70.271,Z 772.146,A -85,B 0,C 180,E1 -28980.443,E2 -28980.443} C_VEL
LIN {X 0,Y 63.64,Z 772.113,A -85,B 0,C 180,E1 -28986.417,E2 -28986.417} C_VEL
LIN {X 0,Y 57.584,Z 771.383,A -85,B 0,C 180,E1 -28994.125,E2 -28994.125} C_VEL
LIN {X 0,Y 52.746,Z 769.88,A -85,B 0,C 180,E1 -29003.557,E2 -29003.557} C_VEL
LIN {X 0,Y 48.679,Z 766.406,A -85,B 0,C 180,E1 -29018.923,E2 -29018.923} C_VEL
LIN {X 0,Y 48.025,Z 761.785,A -85,B 0,C 180,E1 -29034.187,E2 -29034.187} C_VEL
LIN {X 0,Y 49.794,Z 756.456,A -85,B 0,C 180,E1 -29047.103,E2 -29047.103} C_VEL
LIN {X 0,Y 53.133,Z 749.864,A -85,B 0,C 180,E1 -29058.567,E2 -29058.567} C_VEL
LIN {X 0,Y 57.19,Z 743.111,A -85,B 0,C 180,E1 -29066.941,E2 -29066.941} C_VEL
LIN {X 0,Y 62.66,Z 734.152,A -85,B 0,C 180,E1 -29074.718,E2 -29074.718} C_VEL
LIN {X 0,Y 68.762,Z 723.457,A -85,B 0,C 180,E1 -29081.057,E2 -29081.057} C_VEL
LIN {X 0,Y 74.37,Z 712.349,A -85,B 0,C 180,E1 -29085.459,E2 -29085.459} C_VEL
LIN {X 0,Y 79.356,Z 700.568,A -85,B 0,C 180,E1 -29088.733,E2 -29088.733} C_VEL
LIN {X 0,Y 83.647,Z 687.849,A -85,B 0,C 180,E1 -29091.162,E2 -29091.162} C_VEL
LIN {X 0,Y 86.883,Z 674.692,A -85,B 0,C 180,E1 -29092.865,E2 -29092.865} C_VEL
LIN {X 0,Y 89.153,Z 661.281,A -85,B 0,C 180,E1 -29093.872,E2 -29093.872} C_VEL
LIN {X 0,Y 91.96,Z 638.453,A -85,B 0,C 180,E1 -29095.159,E2 -29095.159} C_VEL
LIN {X 0,Y 87.815,Z 628.04,A -85,B 0,C 180,E1 -29100.212,E2 -29100.212} C_VEL
LIN {X 0,Y 83.369,Z 618.989,A -85,B 0,C 180,E1 -29106.452,E2 -29106.452} C_VEL
LIN {X 0,Y 80.303,Z 613.501,A -85,B 0,C 180,E1 -29111.844,E2 -29111.844} C_VEL
LIN {X 0,Y 78.528,Z 610.483,A -85,B 0,C 180,E1 -29115.55,E2 -29115.55} C_VEL
LIN {X 0,Y 76.358,Z 606.792,A -85,B 0,C 180,E1 -29121.364,E2 -29121.364} C_VEL
LIN {X 0,Y 74.422,Z 603.874,A -85,B 0,C 180,E1 -29129.107,E2 -29129.107} C_VEL
LIN {X 0,Y 74.066,Z 602.366,A -85,B 0,C 180,E1 -29132.159,E2 -29132.159} C_VEL
LIN {X 0,Y 73.652,Z 602.128,A -85,B 0,C 180,E1 -29143.368,E2 -29143.368} C_VEL
LIN {X 0,Y 74.647,Z 602.427,A -85,B 0,C 180,E1 -29150.362,E2 -29150.362} C_VEL
LIN {X 0,Y 76.948,Z 606.796,A -85,B 0,C 180,E1 -29159.573,E2 -29159.573} C_VEL
LIN {X 0,Y 79.197,Z 611.097,A -85,B 0,C 180,E1 -29165.248,E2 -29165.248} C_VEL
LIN {X 0,Y 81.963,Z 616.271,A -85,B 0,C 180,E1 -29170.709,E2 -29170.709} C_VEL
LIN {X 0,Y 85.882,Z 624.449,A -85,B 0,C 180,E1 -29176.808,E2 -29176.808} C_VEL
LIN {X 0,Y 88.934,Z 631.972,A -85,B 0,C 180,E1 -29180.953,E2 -29180.953} C_VEL
LIN {X 0,Y 91.683,Z 642.526,A -85,B 0,C 180,E1 -29184.73,E2 -29184.73} C_VEL
LIN {X 0,Y 87.894,Z 672.742,A -85,B 0,C 180,E1 -29186.646,E2 -29186.646} C_VEL
LIN {X 0,Y 85.034,Z 685.685,A -85,B 0,C 180,E1 -29187.942,E2 -29187.942} C_VEL
LIN {X 0,Y 81.1,Z 698.453,A -85,B 0,C 180,E1 -29189.923,E2 -29189.923} C_VEL
LIN {X 0,Y 76.282,Z 710.648,A -85,B 0,C 180,E1 -29192.773,E2 -29192.773} C_VEL
LIN {X 0,Y 71.137,Z 721.609,A -85,B 0,C 180,E1 -29196.501,E2 -29196.501} C_VEL
LIN {X 0,Y 65.592,Z 731.698,A -85,B 0,C 180,E1 -29201.394,E2 -29201.394} C_VEL
LIN {X 0,Y 60.175,Z 740.776,A -85,B 0,C 180,E1 -29207.8,E2 -29207.8} C_VEL
LIN {X 0,Y 54.77,Z 749.619,A -85,B 0,C 180,E1 -29216.939,E2 -29216.939} C_VEL
LIN {X 0,Y 50.984,Z 756.69,A -85,B 0,C 180,E1 -29227.711,E2 -29227.711} C_VEL
LIN {X 0,Y 49.247,Z 761.461,A -85,B 0,C 180,E1 -29237.627,E2 -29237.627} C_VEL
LIN {X 0,Y 48.807,Z 765.983,A -85,B 0,C 180,E1 -29249.988,E2 -29249.988} C_VEL
LIN {X 0,Y 48.901,Z 768.277,A -85,B 0,C 180,E1 -29258.251,E2 -29258.251} C_VEL
LIN {X 0,Y 51.406,Z 771.566,A -85,B 0,C 180,E1 -29274.201,E2 -29274.201} C_VEL
LIN {X 0,Y 57.285,Z 773.392,A -85,B 0,C 180,E1 -29287.824,E2 -29287.824} C_VEL
LIN {X 0,Y 65.973,Z 773.777,A -85,B 0,C 180,E1 -29298.205,E2 -29298.205} C_VEL
LIN {X 0,Y 76.392,Z 772.754,A -85,B 0,C 180,E1 -29305.878,E2 -29305.878} C_VEL
LIN {X 0,Y 87.827,Z 770.33,A -85,B 0,C 180,E1 -29311.655,E2 -29311.655} C_VEL
LIN {X 0,Y 96.962,Z 767.504,A -85,B 0,C 180,E1 -29314.947,E2 -29314.947} C_VEL
LIN {X 0,Y 106.46,Z 763.755,A -85,B 0,C 180,E1 -29317.535,E2 -29317.535} C_VEL
LIN {X 0,Y 115.887,Z 759.139,A -85,B 0,C 180,E1 -29319.694,E2 -29319.694} C_VEL
LIN {X 0,Y 119.382,Z 757.204,A -85,B 0,C 180,E1 -29320.361,E2 -29320.361} C_VEL
LIN {X 0,Y 118.672,Z 757.568,A -85,B 0,C 180,E1 -29321.344,E2 -29321.344} C_VEL
LIN {X 0,Y 107.318,Z 763.087,A -85,B 0,C 180,E1 -29323.927,E2 -29323.927} C_VEL
LIN {X 0,Y 95.969,Z 767.293,A -85,B 0,C 180,E1 -29327.307,E2 -29327.307} C_VEL
LIN {X 0,Y 83.844,Z 770.372,A -85,B 0,C 180,E1 -29332.155,E2 -29332.155} C_VEL
LIN {X 0,Y 78.752,Z 771.303,A -85,B 0,C 180,E1 -29334.203,E2 -29334.203} C_VEL
LIN {X 0,Y 69.569,Z 772.219,A -85,B 0,C 180,E1 -29337.035,E2 -29337.035} C_VEL
LIN {X 0,Y 60.6,Z 772.35,A -85,B 0,C 180,E1 -29340.74,E2 -29340.74} C_VEL
LIN {X 0,Y 56.042,Z 771.977,A -85,B 0,C 180,E1 -29344.404,E2 -29344.404} C_VEL
LIN {X 0,Y 47.596,Z 770.109,A -85,B 0,C 180,E1 -29357.172,E2 -29357.172} C_VEL
LIN {X 0,Y 42.274,Z 766.706,A -85,B 0,C 180,E1 -29373.799,E2 -29373.799} C_VEL
LIN {X 0,Y 40.864,Z 763.549,A -85,B 0,C 180,E1 -29386.552,E2 -29386.552} C_VEL
LIN {X 0,Y 41.721,Z 758.505,A -85,B 0,C 180,E1 -29402.419,E2 -29402.419} C_VEL
LIN {X 0,Y 44.759,Z 752.311,A -85,B 0,C 180,E1 -29416.391,E2 -29416.391} C_VEL
LIN {X 0,Y 49.966,Z 744.196,A -85,B 0,C 180,E1 -29428.701,E2 -29428.701} C_VEL
LIN {X 0,Y 55.696,Z 735.544,A -85,B 0,C 180,E1 -29437.26,E2 -29437.26} C_VEL
LIN {X 0,Y 62.008,Z 725.422,A -85,B 0,C 180,E1 -29443.845,E2 -29443.845} C_VEL
LIN {X 0,Y 68.314,Z 713.99,A -85,B 0,C 180,E1 -29448.762,E2 -29448.762} C_VEL
LIN {X 0,Y 73.253,Z 703.4,A -85,B 0,C 180,E1 -29451.833,E2 -29451.833} C_VEL
LIN {X 0,Y 78.081,Z 690.331,A -85,B 0,C 180,E1 -29454.501,E2 -29454.501} C_VEL
LIN {X 0,Y 81.58,Z 677.818,A -85,B 0,C 180,E1 -29456.188,E2 -29456.188} C_VEL
LIN {X 0,Y 84.265,Z 663.899,A -85,B 0,C 180,E1 -29457.286,E2 -29457.286} C_VEL
LIN {X 0,Y 87.176,Z 641.257,A -85,B 0,C 180,E1 -29458.556,E2 -29458.556} C_VEL
LIN {X 0,Y 86.778,Z 639.6,A -85,B 0,C 180,E1 -29459.189,E2 -29459.189} C_VEL
LIN {X 0,Y 84.119,Z 632.542,A -85,B 0,C 180,E1 -29462.965,E2 -29462.965} C_VEL
LIN {X 0,Y 80.101,Z 623.618,A -85,B 0,C 180,E1 -29469.623,E2 -29469.623} C_VEL
LIN {X 0,Y 77.065,Z 617.769,A -85,B 0,C 180,E1 -29476.033,E2 -29476.033} C_VEL
LIN {X 0,Y 74.708,Z 613.397,A -85,B 0,C 180,E1 -29483,E2 -29483} C_VEL
LIN {X 0,Y 73.046,Z 610.467,A -85,B 0,C 180,E1 -29490.855,E2 -29490.855} C_VEL
LIN {X 0,Y 72.871,Z 609.443,A -85,B 0,C 180,E1 -29492.927,E2 -29492.927} C_VEL
LIN {X 0,Y 72.731,Z 609.18,A -85,B 0,C 180,E1 -29505.113,E2 -29505.113} C_VEL
LIN {X 0,Y 73.394,Z 609.438,A -85,B 0,C 180,E1 -29509.58,E2 -29509.58} C_VEL
LIN {X 0,Y 75.209,Z 613.369,A -85,B 0,C 180,E1 -29517.886,E2 -29517.886} C_VEL
LIN {X 0,Y 77.062,Z 617.385,A -85,B 0,C 180,E1 -29523.33,E2 -29523.33} C_VEL
LIN {X 0,Y 79.421,Z 622.196,A -85,B 0,C 180,E1 -29528.563,E2 -29528.563} C_VEL
LIN {X 0,Y 82.652,Z 629.772,A -85,B 0,C 180,E1 -29534.421,E2 -29534.421} C_VEL
LIN {X 0,Y 85.167,Z 636.446,A -85,B 0,C 180,E1 -29538.269,E2 -29538.269} C_VEL
LIN {X 0,Y 86.99,Z 644.219,A -85,B 0,C 180,E1 -29541.287,E2 -29541.287} C_VEL
LIN {X 0,Y 83.251,Z 672.653,A -85,B 0,C 180,E1 -29543.059,E2 -29543.059} C_VEL
LIN {X 0,Y 80.076,Z 686.334,A -85,B 0,C 180,E1 -29544.399,E2 -29544.399} C_VEL
LIN {X 0,Y 76.327,Z 697.847,A -85,B 0,C 180,E1 -29546.12,E2 -29546.12} C_VEL
LIN {X 0,Y 71.992,Z 708.592,A -85,B 0,C 180,E1 -29548.511,E2 -29548.511} C_VEL
LIN {X 0,Y 65.802,Z 721.133,A -85,B 0,C 180,E1 -29552.609,E2 -29552.609} C_VEL
LIN {X 0,Y 59.871,Z 731.282,A -85,B 0,C 180,E1 -29557.579,E2 -29557.579} C_VEL
LIN {X 0,Y 54.02,Z 740.368,A -85,B 0,C 180,E1 -29564.297,E2 -29564.297} C_VEL
LIN {X 0,Y 48.098,Z 749.207,A -85,B 0,C 180,E1 -29574.22,E2 -29574.22} C_VEL
LIN {X 0,Y 43.963,Z 756.304,A -85,B 0,C 180,E1 -29586.429,E2 -29586.429} C_VEL
LIN {X 0,Y 41.943,Z 761.919,A -85,B 0,C 180,E1 -29600.34,E2 -29600.34} C_VEL
LIN {X 0,Y 41.773,Z 764.932,A -85,B 0,C 180,E1 -29609.986,E2 -29609.986} C_VEL
LIN {X 0,Y 41.941,Z 767.374,A -85,B 0,C 180,E1 -29619.632,E2 -29619.632} C_VEL
LIN {X 0,Y 42.986,Z 769.366,A -85,B 0,C 180,E1 -29629.072,E2 -29629.072} C_VEL
LIN {X 0,Y 48.061,Z 772.1,A -85,B 0,C 180,E1 -29645.782,E2 -29645.782} C_VEL
LIN {X 0,Y 56.426,Z 773.425,A -85,B 0,C 180,E1 -29658.343,E2 -29658.343} C_VEL
LIN {X 0,Y 66.914,Z 773.378,A -85,B 0,C 180,E1 -29667.149,E2 -29667.149} C_VEL
LIN {X 0,Y 78.885,Z 771.832,A -85,B 0,C 180,E1 -29673.545,E2 -29673.545} C_VEL
LIN {X 0,Y 90.981,Z 768.987,A -85,B 0,C 180,E1 -29677.948,E2 -29677.948} C_VEL
LIN {X 0,Y 98.821,Z 766.477,A -85,B 0,C 180,E1 -29679.985,E2 -29679.985} C_VEL
LIN {X 0,Y 101.127,Z 765.577,A -85,B 0,C 180,E1 -29681.252,E2 -29681.252} C_VEL
LIN {X 0,Y 91.165,Z 768.682,A -85,B 0,C 180,E1 -29683.993,E2 -29683.993} C_VEL
LIN {X 0,Y 78.874,Z 771.259,A -85,B 0,C 180,E1 -29688.523,E2 -29688.523} C_VEL
LIN {X 0,Y 68.366,Z 772.341,A -85,B 0,C 180,E1 -29694.097,E2 -29694.097} C_VEL
LIN {X 0,Y 60.473,Z 772.349,A -85,B 0,C 180,E1 -29699.997,E2 -29699.997} C_VEL
LIN {X 0,Y 56.042,Z 771.977,A -85,B 0,C 180,E1 -29704.404,E2 -29704.404} C_VEL
LIN {X 0,Y 51.764,Z 771.394,A -85,B 0,C 180,E1 -29708.678,E2 -29708.678} C_VEL
LIN {X 0,Y 44.072,Z 769.754,A -85,B 0,C 180,E1 -29715.915,E2 -29715.915} C_VEL
LIN {X 0,Y 38.496,Z 767.889,A -85,B 0,C 180,E1 -29723.414,E2 -29723.414} C_VEL
LIN {X 0,Y 35.561,Z 766.172,A -85,B 0,C 180,E1 -29730.972,E2 -29730.972} C_VEL
LIN {X 0,Y 34.979,Z 765.515,A -85,B 0,C 180,E1 -29733.889,E2 -29733.889} C_VEL
LIN {X 0,Y 33.773,Z 761.515,A -85,B 0,C 180,E1 -29751.393,E2 -29751.393} C_VEL
LIN {X 0,Y 35.871,Z 755.604,A -85,B 0,C 180,E1 -29770.703,E2 -29770.703} C_VEL
LIN {X 0,Y 39.957,Z 749.097,A -85,B 0,C 180,E1 -29784.974,E2 -29784.974} C_VEL
LIN {X 0,Y 45.993,Z 740.805,A -85,B 0,C 180,E1 -29796.593,E2 -29796.593} C_VEL
LIN {X 0,Y 52.186,Z 732.159,A -85,B 0,C 180,E1 -29804.203,E2 -29804.203} C_VEL
LIN {X 0,Y 58.844,Z 721.771,A -85,B 0,C 180,E1 -29810.093,E2 -29810.093} C_VEL
LIN {X 0,Y 64.778,Z 711.163,A -85,B 0,C 180,E1 -29814.017,E2 -29814.017} C_VEL
LIN {X 0,Y 69.891,Z 700.158,A -85,B 0,C 180,E1 -29816.83,E2 -29816.83} C_VEL
LIN {X 0,Y 74.472,Z 687.579,A -85,B 0,C 180,E1 -29819.025,E2 -29819.025} C_VEL
LIN {X 0,Y 77.992,Z 674.386,A -85,B 0,C 180,E1 -29820.564,E2 -29820.564} C_VEL
LIN {X 0,Y 80.422,Z 660.88,A -85,B 0,C 180,E1 -29821.42,E2 -29821.42} C_VEL
LIN {X 0,Y 82.691,Z 643.044,A -85,B 0,C 180,E1 -29822.46,E2 -29822.46} C_VEL
LIN {X 0,Y 80.666,Z 637.195,A -85,B 0,C 180,E1 -29825.847,E2 -29825.847} C_VEL
LIN {X 0,Y 77.463,Z 629.229,A -85,B 0,C 180,E1 -29832.151,E2 -29832.151} C_VEL
LIN {X 0,Y 74.757,Z 623.419,A -85,B 0,C 180,E1 -29838.85,E2 -29838.85} C_VEL
LIN {X 0,Y 73.102,Z 619.995,A -85,B 0,C 180,E1 -29844.775,E2 -29844.775} C_VEL
LIN {X 0,Y 71.703,Z 616.798,A -85,B 0,C 180,E1 -29853.225,E2 -29853.225} C_VEL
LIN {X 0,Y 71.591,Z 616.299,A -85,B 0,C 180,E1 -29854.948,E2 -29854.948} C_VEL
LIN {X 0,Y 72.1,Z 616.279,A -85,B 0,C 180,E1 -29868.345,E2 -29868.345} C_VEL
LIN {X 0,Y 73.508,Z 619.894,A -85,B 0,C 180,E1 -29876.014,E2 -29876.014} C_VEL
LIN {X 0,Y 75.226,Z 624.151,A -85,B 0,C 180,E1 -29881.902,E2 -29881.902} C_VEL
LIN {X 0,Y 77.102,Z 628.491,A -85,B 0,C 180,E1 -29886.568,E2 -29886.568} C_VEL
LIN {X 0,Y 79.582,Z 635.057,A -85,B 0,C 180,E1 -29891.843,E2 -29891.843} C_VEL
LIN {X 0,Y 81.467,Z 640.725,A -85,B 0,C 180,E1 -29895.289,E2 -29895.289} C_VEL
LIN {X 0,Y 82.609,Z 646.061,A -85,B 0,C 180,E1 -29897.511,E2 -29897.511} C_VEL
LIN {X 0,Y 78.967,Z 672.309,A -85,B 0,C 180,E1 -29899.056,E2 -29899.056} C_VEL
LIN {X 0,Y 75.623,Z 686.173,A -85,B 0,C 180,E1 -29900.334,E2 -29900.334} C_VEL
LIN {X 0,Y 71.188,Z 699.021,A -85,B 0,C 180,E1 -29902.229,E2 -29902.229} C_VEL
LIN {X 0,Y 66.396,Z 709.893,A -85,B 0,C 180,E1 -29904.615,E2 -29904.615} C_VEL
LIN {X 0,Y 60.799,Z 720.527,A -85,B 0,C 180,E1 -29908.081,E2 -29908.081} C_VEL
LIN {X 0,Y 54.478,Z 730.709,A -85,B 0,C 180,E1 -29912.996,E2 -29912.996} C_VEL
LIN {X 0,Y 48.129,Z 739.862,A -85,B 0,C 180,E1 -29919.93,E2 -29919.93} C_VEL
LIN {X 0,Y 41.583,Z 748.742,A -85,B 0,C 180,E1 -29930.652,E2 -29930.652} C_VEL
LIN {X 0,Y 36.968,Z 755.892,A -85,B 0,C 180,E1 -29944.658,E2 -29944.658} C_VEL
LIN {X 0,Y 34.995,Z 760.682,A -85,B 0,C 180,E1 -29958.398,E2 -29958.398} C_VEL
LIN {X 0,Y 34.742,Z 763.882,A -85,B 0,C 180,E1 -29969.983,E2 -29969.983} C_VEL
LIN {X 0,Y 35.527,Z 767.533,A -85,B 0,C 180,E1 -29987.244,E2 -29987.244} C_VEL
LIN {X 0,Y 38.925,Z 770.19,A -85,B 0,C 180,E1 -30002.778,E2 -30002.778} C_VEL
LIN {X 0,Y 46.871,Z 772.464,A -85,B 0,C 180,E1 -30018.547,E2 -30018.547} C_VEL
LIN {X 0,Y 57.473,Z 773.316,A -85,B 0,C 180,E1 -30028.848,E2 -30028.848} C_VEL
LIN {X 0,Y 69.415,Z 772.806,A -85,B 0,C 180,E1 -30035.653,E2 -30035.653} C_VEL
LIN {X 0,Y 82.05,Z 770.91,A -85,B 0,C 180,E1 -30040.402,E2 -30040.402} C_VEL
LIN {X 0,Y 81.324,Z 770.983,A -85,B 0,C 180,E1 -30041.893,E2 -30041.893} C_VEL
LIN {X 0,Y 72.752,Z 772.139,A -85,B 0,C 180,E1 -30044.988,E2 -30044.988} C_VEL
LIN {X 0,Y 64.424,Z 772.65,A -85,B 0,C 180,E1 -30049.004,E2 -30049.004} C_VEL
LIN {X 0,Y 56.503,Z 772.513,A -85,B 0,C 180,E1 -30054.201,E2 -30054.201} C_VEL
LIN {X 0,Y 49.193,Z 771.683,A -85,B 0,C 180,E1 -30061.006,E2 -30061.006} C_VEL
LIN {X 0,Y 40.109,Z 769.204,A -85,B 0,C 180,E1 -30075.536,E2 -30075.536} C_VEL
LIN {X 0,Y 34.979,Z 765.515,A -85,B 0,C 180,E1 -30093.889,E2 -30093.889} C_VEL
LIN {X 0,Y 33.354,Z 763.498,A -85,B 0,C 180,E1 -30102.797,E2 -30102.797} C_VEL
LIN {X 0,Y 31.584,Z 761.156,A -85,B 0,C 180,E1 -30111.949,E2 -30111.949} C_VEL
LIN {X 0,Y 29.931,Z 754.654,A -85,B 0,C 180,E1 -30135.026,E2 -30135.026} C_VEL
LIN {X 0,Y 31.5,Z 751.431,A -85,B 0,C 180,E1 -30143.982,E2 -30143.982} C_VEL
LIN {X 0,Y 37.753,Z 743.692,A -85,B 0,C 180,E1 -30158.2,E2 -30158.2} C_VEL
LIN {X 0,Y 45.236,Z 734.235,A -85,B 0,C 180,E1 -30168.116,E2 -30168.116} C_VEL
LIN {X 0,Y 51.945,Z 724.896,A -85,B 0,C 180,E1 -30173.959,E2 -30173.959} C_VEL
LIN {X 0,Y 58.292,Z 714.702,A -85,B 0,C 180,E1 -30178.033,E2 -30178.033} C_VEL
LIN {X 0,Y 64.569,Z 702.488,A -85,B 0,C 180,E1 -30181.146,E2 -30181.146} C_VEL
LIN {X 0,Y 69.763,Z 689.469,A -85,B 0,C 180,E1 -30183.402,E2 -30183.402} C_VEL
LIN {X 0,Y 73.502,Z 676.778,A -85,B 0,C 180,E1 -30184.773,E2 -30184.773} C_VEL
LIN {X 0,Y 76.19,Z 663.384,A -85,B 0,C 180,E1 -30185.627,E2 -30185.627} C_VEL
LIN {X 0,Y 78.608,Z 645.555,A -85,B 0,C 180,E1 -30186.562,E2 -30186.562} C_VEL
LIN {X 0,Y 76.584,Z 639.39,A -85,B 0,C 180,E1 -30190.861,E2 -30190.861} C_VEL
LIN {X 0,Y 74.618,Z 634.219,A -85,B 0,C 180,E1 -30195.553,E2 -30195.553} C_VEL
LIN {X 0,Y 72.779,Z 629.595,A -85,B 0,C 180,E1 -30201.243,E2 -30201.243} C_VEL
LIN {X 0,Y 71.485,Z 626.498,A -85,B 0,C 180,E1 -30206.799,E2 -30206.799} C_VEL
LIN {X 0,Y 70.457,Z 623.275,A -85,B 0,C 180,E1 -30215.793,E2 -30215.793} C_VEL
LIN {X 0,Y 70.88,Z 623.308,A -85,B 0,C 180,E1 -30227.518,E2 -30227.518} C_VEL
LIN {X 0,Y 71.915,Z 626.494,A -85,B 0,C 180,E1 -30234.198,E2 -30234.198} C_VEL
LIN {X 0,Y 73.187,Z 630.227,A -85,B 0,C 180,E1 -30239.551,E2 -30239.551} C_VEL
LIN {X 0,Y 74.651,Z 634.255,A -85,B 0,C 180,E1 -30244.005,E2 -30244.005} C_VEL
LIN {X 0,Y 76.725,Z 640.461,A -85,B 0,C 180,E1 -30249.162,E2 -30249.162} C_VEL
LIN {X 0,Y 78.029,Z 645.079,A -85,B 0,C 180,E1 -30252.097,E2 -30252.097} C_VEL
LIN {X 0,Y 78.529,Z 647.941,A -85,B 0,C 180,E1 -30253.368,E2 -30253.368} C_VEL
LIN {X 0,Y 74.869,Z 672.793,A -85,B 0,C 180,E1 -30254.72,E2 -30254.72} C_VEL
LIN {X 0,Y 71.669,Z 685.52,A -85,B 0,C 180,E1 -30255.768,E2 -30255.768} C_VEL
LIN {X 0,Y 67.216,Z 698.114,A -85,B 0,C 180,E1 -30257.402,E2 -30257.402} C_VEL
LIN {X 0,Y 62.438,Z 708.677,A -85,B 0,C 180,E1 -30259.475,E2 -30259.475} C_VEL
LIN {X 0,Y 55.818,Z 720.6,A -85,B 0,C 180,E1 -30263.04,E2 -30263.04} C_VEL
LIN {X 0,Y 49.504,Z 730.117,A -85,B 0,C 180,E1 -30267.44,E2 -30267.44} C_VEL
LIN {X 0,Y 42.577,Z 739.347,A -85,B 0,C 180,E1 -30274.355,E2 -30274.355} C_VEL
LIN {X 0,Y 35.277,Z 748.265,A -85,B 0,C 180,E1 -30285.769,E2 -30285.769} C_VEL
LIN {X 0,Y 30.03,Z 755.438,A -85,B 0,C 180,E1 -30302.07,E2 -30302.07} C_VEL
LIN {X 0,Y 27.719,Z 761.117,A -85,B 0,C 180,E1 -30322.696,E2 -30322.696} C_VEL
LIN {X 0,Y 27.81,Z 764.111,A -85,B 0,C 180,E1 -30337.238,E2 -30337.238} C_VEL
LIN {X 0,Y 29.998,Z 767.616,A -85,B 0,C 180,E1 -30357.919,E2 -30357.919} C_VEL
LIN {X 0,Y 37.486,Z 770.842,A -85,B 0,C 180,E1 -30378.561,E2 -30378.561} C_VEL
LIN {X 0,Y 48.164,Z 772.652,A -85,B 0,C 180,E1 -30391.08,E2 -30391.08} C_VEL
LIN {X 0,Y 60.404,Z 773.082,A -85,B 0,C 180,E1 -30398.533,E2 -30398.533} C_VEL
LIN {X 0,Y 65.766,Z 772.835,A -85,B 0,C 180,E1 -30401.298,E2 -30401.298} C_VEL
LIN {X 0,Y 56.525,Z 772.806,A -85,B 0,C 180,E1 -30405.598,E2 -30405.598} C_VEL
LIN {X 0,Y 47.802,Z 772.046,A -85,B 0,C 180,E1 -30411.541,E2 -30411.541} C_VEL
LIN {X 0,Y 39.727,Z 770.533,A -85,B 0,C 180,E1 -30419.995,E2 -30419.995} C_VEL
LIN {X 0,Y 33,Z 768.209,A -85,B 0,C 180,E1 -30432.29,E2 -30432.29} C_VEL
LIN {X 0,Y 28.266,Z 764.968,A -85,B 0,C 180,E1 -30449.815,E2 -30449.815} C_VEL
LIN {X 0,Y 26.721,Z 760.617,A -85,B 0,C 180,E1 -30472.085,E2 -30472.085} C_VEL
LIN {X 0,Y 29.156,Z 754.834,A -85,B 0,C 180,E1 -30494.593,E2 -30494.593} C_VEL
LIN {X 0,Y 31.5,Z 751.431,A -85,B 0,C 180,E1 -30503.982,E2 -30503.982} C_VEL
LIN {X 0,Y 33.525,Z 748.067,A -85,B 0,C 180,E1 -30511.676,E2 -30511.676} C_VEL
LIN {X 0,Y 36.262,Z 741.924,A -85,B 0,C 180,E1 -30523.693,E2 -30523.693} C_VEL
LIN {X 0,Y 39.867,Z 735.211,A -85,B 0,C 180,E1 -30533.412,E2 -30533.412} C_VEL
LIN {X 0,Y 42.938,Z 730.854,A -85,B 0,C 180,E1 -30537.132,E2 -30537.132} C_VEL
LIN {X 0,Y 50.678,Z 720.181,A -85,B 0,C 180,E1 -30542.163,E2 -30542.163} C_VEL
LIN {X 0,Y 57.664,Z 708.541,A -85,B 0,C 180,E1 -30545.387,E2 -30545.387} C_VEL
LIN {X 0,Y 63.614,Z 696.001,A -85,B 0,C 180,E1 -30547.671,E2 -30547.671} C_VEL
LIN {X 0,Y 67.814,Z 684.593,A -85,B 0,C 180,E1 -30549.011,E2 -30549.011} C_VEL
LIN {X 0,Y 71.316,Z 671.106,A -85,B 0,C 180,E1 -30550.089,E2 -30550.089} C_VEL
LIN {X 0,Y 74.471,Z 651.888,A -85,B 0,C 180,E1 -30550.845,E2 -30550.845} C_VEL
LIN {X 0,Y 74.915,Z 648.044,A -85,B 0,C 180,E1 -30551.165,E2 -30551.165} C_VEL
LIN {X 0,Y 72.515,Z 640.414,A -85,B 0,C 180,E1 -30557.74,E2 -30557.74} C_VEL
LIN {X 0,Y 70.987,Z 635.844,A -85,B 0,C 180,E1 -30563.561,E2 -30563.561} C_VEL
LIN {X 0,Y 70.011,Z 633.148,A -85,B 0,C 180,E1 -30568.561,E2 -30568.561} C_VEL
LIN {X 0,Y 69.348,Z 630.398,A -85,B 0,C 180,E1 -30576.089,E2 -30576.089} C_VEL
LIN {X 0,Y 69.682,Z 630.266,A -85,B 0,C 180,E1 -30586.632,E2 -30586.632} C_VEL
LIN {X 0,Y 70.388,Z 633.122,A -85,B 0,C 180,E1 -30592.416,E2 -30592.416} C_VEL
LIN {X 0,Y 71.339,Z 636.565,A -85,B 0,C 180,E1 -30597.372,E2 -30597.372} C_VEL
LIN {X 0,Y 72.318,Z 639.895,A -85,B 0,C 180,E1 -30601.142,E2 -30601.142} C_VEL
LIN {X 0,Y 73.914,Z 645.567,A -85,B 0,C 180,E1 -30606.033,E2 -30606.033} C_VEL
LIN {X 0,Y 74.84,Z 649.487,A -85,B 0,C 180,E1 -30608.617,E2 -30608.617} C_VEL
LIN {X 0,Y 74.621,Z 652.15,A -85,B 0,C 180,E1 -30608.981,E2 -30608.981} C_VEL
LIN {X 0,Y 71.348,Z 672.787,A -85,B 0,C 180,E1 -30609.882,E2 -30609.882} C_VEL
LIN {X 0,Y 67.885,Z 686.034,A -85,B 0,C 180,E1 -30610.825,E2 -30610.825} C_VEL
LIN {X 0,Y 63.242,Z 698.445,A -85,B 0,C 180,E1 -30612.206,E2 -30612.206} C_VEL
LIN {X 0,Y 57.969,Z 709.375,A -85,B 0,C 180,E1 -30614.056,E2 -30614.056} C_VEL
LIN {X 0,Y 51.458,Z 720.424,A -85,B 0,C 180,E1 -30617.015,E2 -30617.015} C_VEL
LIN {X 0,Y 45.1,Z 729.415,A -85,B 0,C 180,E1 -30620.738,E2 -30620.738} C_VEL
LIN {X 0,Y 37.559,Z 738.733,A -85,B 0,C 180,E1 -30627.242,E2 -30627.242} C_VEL
LIN {X 0,Y 29.363,Z 747.692,A -85,B 0,C 180,E1 -30638.901,E2 -30638.901} C_VEL
LIN {X 0,Y 23.2,Z 754.921,A -85,B 0,C 180,E1 -30657.957,E2 -30657.957} C_VEL
LIN {X 0,Y 20.742,Z 759.769,A -85,B 0,C 180,E1 -30680.218,E2 -30680.218} C_VEL
LIN {X 0,Y 20.875,Z 762.977,A -85,B 0,C 180,E1 -30699.663,E2 -30699.663} C_VEL
LIN {X 0,Y 23.993,Z 766.654,A -85,B 0,C 180,E1 -30725.832,E2 -30725.832} C_VEL
LIN {X 0,Y 33.224,Z 770.142,A -85,B 0,C 180,E1 -30747.761,E2 -30747.761} C_VEL
LIN {X 0,Y 38.953,Z 771.318,A -85,B 0,C 180,E1 -30754.403,E2 -30754.403} C_VEL
LIN {X 0,Y 46.169,Z 772.277,A -85,B 0,C 180,E1 -30759.619,E2 -30759.619} C_VEL
LIN {X 0,Y 47.937,Z 772.431,A -85,B 0,C 180,E1 -30761.678,E2 -30761.678} C_VEL
LIN {X 0,Y 35.544,Z 770.233,A -85,B 0,C 180,E1 -30771.241,E2 -30771.241} C_VEL
LIN {X 0,Y 25.11,Z 766.549,A -85,B 0,C 180,E1 -30789.879,E2 -30789.879} C_VEL
LIN {X 0,Y 20.599,Z 763.056,A -85,B 0,C 180,E1 -30811.521,E2 -30811.521} C_VEL
LIN {X 0,Y 20.323,Z 757.674,A -85,B 0,C 180,E1 -30844.626,E2 -30844.626} C_VEL
LIN {X 0,Y 24.119,Z 752.219,A -85,B 0,C 180,E1 -30866.845,E2 -30866.845} C_VEL
LIN {X 0,Y 30.743,Z 744.919,A -85,B 0,C 180,E1 -30883.234,E2 -30883.234} C_VEL
LIN {X 0,Y 38.181,Z 736.616,A -85,B 0,C 180,E1 -30893.035,E2 -30893.035} C_VEL
LIN {X 0,Y 42.938,Z 730.854,A -85,B 0,C 180,E1 -30897.132,E2 -30897.132} C_VEL
LIN {X 0,Y 45.936,Z 726.414,A -85,B 0,C 180,E1 -30900.218,E2 -30900.218} C_VEL
LIN {X 0,Y 49.766,Z 718.662,A -85,B 0,C 180,E1 -30906.028,E2 -30906.028} C_VEL
LIN {X 0,Y 53.452,Z 710.495,A -85,B 0,C 180,E1 -30910.819,E2 -30910.819} C_VEL
LIN {X 0,Y 56.012,Z 705.282,A -85,B 0,C 180,E1 -30912.337,E2 -30912.337} C_VEL
LIN {X 0,Y 61.672,Z 692.899,A -85,B 0,C 180,E1 -30913.858,E2 -30913.858} C_VEL
LIN {X 0,Y 66.383,Z 679.097,A -85,B 0,C 180,E1 -30914.904,E2 -30914.904} C_VEL
LIN {X 0,Y 69.267,Z 666.278,A -85,B 0,C 180,E1 -30915.543,E2 -30915.543} C_VEL
LIN {X 0,Y 71.592,Z 650.989,A -85,B 0,C 180,E1 -30916.076,E2 -30916.076} C_VEL
LIN {X 0,Y 70.172,Z 645.447,A -85,B 0,C 180,E1 -30921.479,E2 -30921.479} C_VEL
LIN {X 0,Y 69.171,Z 641.751,A -85,B 0,C 180,E1 -30926.546,E2 -30926.546} C_VEL
LIN {X 0,Y 68.619,Z 639.787,A -85,B 0,C 180,E1 -30930.333,E2 -30930.333} C_VEL
LIN {X 0,Y 68.224,Z 637.331,A -85,B 0,C 180,E1 -30937.429,E2 -30937.429} C_VEL
LIN {X 0,Y 68.483,Z 637.289,A -85,B 0,C 180,E1 -30945.642,E2 -30945.642} C_VEL
LIN {X 0,Y 68.886,Z 639.604,A -85,B 0,C 180,E1 -30950.336,E2 -30950.336} C_VEL
LIN {X 0,Y 69.963,Z 644.321,A -85,B 0,C 180,E1 -30956.943,E2 -30956.943} C_VEL
LIN {X 0,Y 71.353,Z 650.82,A -85,B 0,C 180,E1 -30962.878,E2 -30962.878} C_VEL
LIN {X 0,Y 71.625,Z 652.232,A -85,B 0,C 180,E1 -30963.885,E2 -30963.885} C_VEL
LIN {X 0,Y 68.266,Z 672.825,A -85,B 0,C 180,E1 -30964.638,E2 -30964.638} C_VEL
LIN {X 0,Y 64.569,Z 686.383,A -85,B 0,C 180,E1 -30965.368,E2 -30965.368} C_VEL
LIN {X 0,Y 59.769,Z 698.668,A -85,B 0,C 180,E1 -30966.401,E2 -30966.401} C_VEL
LIN {X 0,Y 53.275,Z 711.412,A -85,B 0,C 180,E1 -30968.13,E2 -30968.13} C_VEL
LIN {X 0,Y 46.47,Z 721.995,A -85,B 0,C 180,E1 -30970.5,E2 -30970.5} C_VEL
LIN {X 0,Y 38.137,Z 732.624,A -85,B 0,C 180,E1 -30974.595,E2 -30974.595} C_VEL
LIN {X 0,Y 30.114,Z 741.31,A -85,B 0,C 180,E1 -30980.959,E2 -30980.959} C_VEL
LIN {X 0,Y 21.269,Z 749.728,A -85,B 0,C 180,E1 -30994.253,E2 -30994.253} C_VEL
LIN {X 0,Y 14.894,Z 756.47,A -85,B 0,C 180,E1 -31021.8,E2 -31021.8} C_VEL
LIN {X 0,Y 13.649,Z 760.157,A -85,B 0,C 180,E1 -31049.958,E2 -31049.958} C_VEL
LIN {X 0,Y 15,Z 763.157,A -85,B 0,C 180,E1 -31077.896,E2 -31077.896} C_VEL
LIN {X 0,Y 24.015,Z 767.665,A -85,B 0,C 180,E1 -31111.346,E2 -31111.346} C_VEL
LIN {X 0,Y 30.049,Z 769.354,A -85,B 0,C 180,E1 -31119.26,E2 -31119.26} C_VEL
LIN {X 0,Y 29.359,Z 769.108,A -85,B 0,C 180,E1 -31123.169,E2 -31123.169} C_VEL
LIN {X 0,Y 18.998,Z 765.369,A -85,B 0,C 180,E1 -31139.989,E2 -31139.989} C_VEL
LIN {X 0,Y 12.657,Z 759.894,A -85,B 0,C 180,E1 -31184.228,E2 -31184.228} C_VEL
LIN {X 0,Y 15.283,Z 754.592,A -85,B 0,C 180,E1 -31224.607,E2 -31224.607} C_VEL
LIN {X 0,Y 22.514,Z 747.621,A -85,B 0,C 180,E1 -31248.216,E2 -31248.216} C_VEL
LIN {X 0,Y 29.735,Z 740.739,A -85,B 0,C 180,E1 -31258.232,E2 -31258.232} C_VEL
LIN {X 0,Y 38.286,Z 731.438,A -85,B 0,C 180,E1 -31265.025,E2 -31265.025} C_VEL
LIN {X 0,Y 46.105,Z 721.394,A -85,B 0,C 180,E1 -31268.977,E2 -31268.977} C_VEL
LIN {X 0,Y 53.071,Z 710.618,A -85,B 0,C 180,E1 -31271.476,E2 -31271.476} C_VEL
LIN {X 0,Y 56.012,Z 705.282,A -85,B 0,C 180,E1 -31272.337,E2 -31272.337} C_VEL
LIN {X 0,Y 58.346,Z 700.018,A -85,B 0,C 180,E1 -31273.676,E2 -31273.676} C_VEL
LIN {X 0,Y 61.035,Z 691.155,A -85,B 0,C 180,E1 -31277.106,E2 -31277.106} C_VEL
LIN {X 0,Y 63.285,Z 682.021,A -85,B 0,C 180,E1 -31280.115,E2 -31280.115} C_VEL
LIN {X 0,Y 64.681,Z 676.327,A -85,B 0,C 180,E1 -31280.93,E2 -31280.93} C_VEL
LIN {X 0,Y 67.427,Z 663.389,A -85,B 0,C 180,E1 -31281.167,E2 -31281.167} C_VEL
LIN {X 0,Y 68.744,Z 654.767,A -85,B 0,C 180,E1 -31281.33,E2 -31281.33} C_VEL
LIN {X 0,Y 68.734,Z 653.822,A -85,B 0,C 180,E1 -31281.785,E2 -31281.785} C_VEL
LIN {X 0,Y 68.013,Z 649.938,A -85,B 0,C 180,E1 -31286.091,E2 -31286.091} C_VEL
LIN {X 0,Y 67.364,Z 646.718,A -85,B 0,C 180,E1 -31291.429,E2 -31291.429} C_VEL
LIN {X 0,Y 67.132,Z 644.319,A -85,B 0,C 180,E1 -31298.67,E2 -31298.67} C_VEL
LIN {X 0,Y 67.306,Z 644.344,A -85,B 0,C 180,E1 -31304.687,E2 -31304.687} C_VEL
LIN {X 0,Y 67.608,Z 646.993,A -85,B 0,C 180,E1 -31309.678,E2 -31309.678} C_VEL
LIN {X 0,Y 68.195,Z 650.74,A -85,B 0,C 180,E1 -31314.458,E2 -31314.458} C_VEL
LIN {X 0,Y 68.818,Z 654.914,A -85,B 0,C 180,E1 -31318.471,E2 -31318.471} C_VEL
LIN {X 0,Y 65.638,Z 673.546,A -85,B 0,C 180,E1 -31318.985,E2 -31318.985} C_VEL
LIN {X 0,Y 61.946,Z 686.543,A -85,B 0,C 180,E1 -31319.386,E2 -31319.386} C_VEL
LIN {X 0,Y 56.806,Z 699.285,A -85,B 0,C 180,E1 -31320.004,E2 -31320.004} C_VEL
LIN {X 0,Y 50.353,Z 711.504,A -85,B 0,C 180,E1 -31320.939,E2 -31320.939} C_VEL
LIN {X 0,Y 43.093,Z 722.331,A -85,B 0,C 180,E1 -31322.359,E2 -31322.359} C_VEL
LIN {X 0,Y 35.259,Z 731.865,A -85,B 0,C 180,E1 -31324.512,E2 -31324.512} C_VEL
LIN {X 0,Y 26.655,Z 740.602,A -85,B 0,C 180,E1 -31328.467,E2 -31328.467} C_VEL
LIN {X 0,Y 18.261,Z 747.799,A -85,B 0,C 180,E1 -31335.695,E2 -31335.695} C_VEL
LIN {X 0,Y 9.303,Z 754.883,A -85,B 0,C 180,E1 -31360.839,E2 -31360.839} C_VEL
LIN {X 0,Y 6.618,Z 758.732,A -85,B 0,C 180,E1 -31409.913,E2 -31409.913} C_VEL
LIN {X 0,Y 9.419,Z 761.896,A -85,B 0,C 180,E1 -31458.165,E2 -31458.165} C_VEL
LIN {X 0,Y 15.055,Z 764.531,A -85,B 0,C 180,E1 -31478.904,E2 -31478.904} C_VEL
LIN {X 0,Y 14.917,Z 764.466,A -85,B 0,C 180,E1 -31480.319,E2 -31480.319} C_VEL
LIN {X 0,Y 5.977,Z 759.34,A -85,B 0,C 180,E1 -31528.377,E2 -31528.377} C_VEL
LIN {X 0,Y 10.758,Z 752.953,A -85,B 0,C 180,E1 -31609.121,E2 -31609.121} C_VEL
LIN {X 0,Y 20.612,Z 745.288,A -85,B 0,C 180,E1 -31626.701,E2 -31626.701} C_VEL
LIN {X 0,Y 29.057,Z 737.651,A -85,B 0,C 180,E1 -31632.512,E2 -31632.512} C_VEL
LIN {X 0,Y 37.945,Z 728.066,A -85,B 0,C 180,E1 -31635.887,E2 -31635.887} C_VEL
LIN {X 0,Y 46.176,Z 717.161,A -85,B 0,C 180,E1 -31637.995,E2 -31637.995} C_VEL
LIN {X 0,Y 53.348,Z 705.394,A -85,B 0,C 180,E1 -31639.27,E2 -31639.27} C_VEL
LIN {X 0,Y 58.796,Z 693.864,A -85,B 0,C 180,E1 -31640.109,E2 -31640.109} C_VEL
LIN {X 0,Y 63.687,Z 680.062,A -85,B 0,C 180,E1 -31640.746,E2 -31640.746} C_VEL
LIN {X 0,Y 64.681,Z 676.327,A -85,B 0,C 180,E1 -31640.93,E2 -31640.93} C_VEL
LIN {X 0,Y 66.14,Z 669.372,A -85,B 0,C 180,E1 -31641.629,E2 -31641.629} C_VEL
LIN {X 0,Y 66.707,Z 663.992,A -85,B 0,C 180,E1 -31643.02,E2 -31643.02} C_VEL
LIN {X 0,Y 66.771,Z 660.4,A -85,B 0,C 180,E1 -31644.707,E2 -31644.707} C_VEL
LIN {X 0,Y 66.556,Z 657.264,A -85,B 0,C 180,E1 -31647.308,E2 -31647.308} C_VEL
LIN {X 0,Y 66.469,Z 656.72,A -85,B 0,C 180,E1 -31648.036,E2 -31648.036} C_VEL
LIN {X 0,Y 66.122,Z 653.911,A -85,B 0,C 180,E1 -31652.351,E2 -31652.351} C_VEL
LIN {X 0,Y 66.057,Z 651.31,A -85,B 0,C 180,E1 -31659.28,E2 -31659.28} C_VEL
LIN {X 0,Y 66.155,Z 651.361,A -85,B 0,C 180,E1 -31663.7,E2 -31663.7} C_VEL
LIN {X 0,Y 66.316,Z 654.845,A -85,B 0,C 180,E1 -31669.262,E2 -31669.262} C_VEL
LIN {X 0,Y 66.591,Z 657.817,A -85,B 0,C 180,E1 -31672.641,E2 -31672.641} C_VEL
LIN {X 0,Y 63.744,Z 673.86,A -85,B 0,C 180,E1 -31672.948,E2 -31672.948} C_VEL
LIN {X 0,Y 60.021,Z 686.607,A -85,B 0,C 180,E1 -31672.956,E2 -31672.956} C_VEL
LIN {X 0,Y 54.621,Z 699.716,A -85,B 0,C 180,E1 -31672.993,E2 -31672.993} C_VEL
LIN {X 0,Y 48.691,Z 710.758,A -85,B 0,C 180,E1 -31672.99,E2 -31672.99} C_VEL
LIN {X 0,Y 41.604,Z 721.33,A -85,B 0,C 180,E1 -31673.062,E2 -31673.062} C_VEL
LIN {X 0,Y 33.636,Z 730.98,A -85,B 0,C 180,E1 -31673.104,E2 -31673.104} C_VEL
LIN {X 0,Y 24.777,Z 739.827,A -85,B 0,C 180,E1 -31673.307,E2 -31673.307} C_VEL
LIN {X 0,Y 14.174,Z 748.428,A -85,B 0,C 180,E1 -31672.909,E2 -31672.909} C_VEL
LIN {X 0,Y 7.103,Z 753.173,A -85,B 0,C 180,E1 -31672.243,E2 -31672.243} C_VEL
LIN {X 0,Y 5.671,Z 753.965,A -85,B 0,C 180,E1 -31654.156,E2 -31654.156} C_VEL
LIN {X 0,Y 14.976,Z 747.646,A -85,B 0,C 180,E1 -31647.174,E2 -31647.174} C_VEL
LIN {X 0,Y 25.42,Z 738.945,A -85,B 0,C 180,E1 -31646.44,E2 -31646.44} C_VEL
LIN {X 0,Y 35.025,Z 729.073,A -85,B 0,C 180,E1 -31646.529,E2 -31646.529} C_VEL
LIN {X 0,Y 43.133,Z 718.731,A -85,B 0,C 180,E1 -31646.645,E2 -31646.645} C_VEL
LIN {X 0,Y 50.446,Z 707.186,A -85,B 0,C 180,E1 -31646.73,E2 -31646.73} C_VEL
LIN {X 0,Y 56.112,Z 695.862,A -85,B 0,C 180,E1 -31646.907,E2 -31646.907} C_VEL
LIN {X 0,Y 61.146,Z 682.441,A -85,B 0,C 180,E1 -31646.989,E2 -31646.989} C_VEL
LIN {X 0,Y 64.672,Z 668.776,A -85,B 0,C 180,E1 -31647.139,E2 -31647.139} C_VEL
LIN {X 0,Y 66.556,Z 657.342,A -85,B 0,C 180,E1 -31647.255,E2 -31647.255} C_VEL
LIN {X 0,Y 66.469,Z 656.72,A -85,B 0,C 180,E1 -31648.036,E2 -31648.036} C_VEL
LIN {X 0,Y 66.036,Z 655.526,A -85,B 0,C 180,E1 -31651.289,E2 -31651.289} C_VEL
LIN {X 0,Y 65.607,Z 655.577,A -85,B 0,C 180,E1 -31654.786,E2 -31654.786} C_VEL
LIN {X 0,Y 65.179,Z 657.033,A -85,B 0,C 180,E1 -31659.49,E2 -31659.49} C_VEL
LIN {X 0,Y 64.932,Z 660.92,A -85,B 0,C 180,E1 -31666.275,E2 -31666.275} C_VEL
LIN {X 0,Y 64.934,Z 661.108,A -85,B 0,C 180,E1 -31666.533,E2 -31666.533} C_VEL
LIN {X 0,Y 62.469,Z 674.253,A -85,B 0,C 180,E1 -31666.555,E2 -31666.555} C_VEL
LIN {X 0,Y 58.473,Z 687.592,A -85,B 0,C 180,E1 -31666.139,E2 -31666.139} C_VEL
LIN {X 0,Y 53.182,Z 700.284,A -85,B 0,C 180,E1 -31665.489,E2 -31665.489} C_VEL
LIN {X 0,Y 46.516,Z 712.435,A -85,B 0,C 180,E1 -31664.45,E2 -31664.45} C_VEL
LIN {X 0,Y 38.646,Z 723.776,A -85,B 0,C 180,E1 -31662.743,E2 -31662.743} C_VEL
LIN {X 0,Y 34.237,Z 729.199,A -85,B 0,C 180,E1 -31661.351,E2 -31661.351} C_VEL
LIN {X 0,Y 32.753,Z 730.845,A -85,B 0,C 180,E1 -31658.862,E2 -31658.862} C_VEL
LIN {X 0,Y 41.222,Z 720.269,A -85,B 0,C 180,E1 -31656.438,E2 -31656.438} C_VEL
LIN {X 0,Y 48.971,Z 708.109,A -85,B 0,C 180,E1 -31654.925,E2 -31654.925} C_VEL
LIN {X 0,Y 55.205,Z 695.644,A -85,B 0,C 180,E1 -31654.134,E2 -31654.134} C_VEL
LIN {X 0,Y 60.26,Z 681.907,A -85,B 0,C 180,E1 -31653.613,E2 -31653.613} C_VEL
LIN {X 0,Y 63.674,Z 668.337,A -85,B 0,C 180,E1 -31653.389,E2 -31653.389} C_VEL
LIN {X 0,Y 64.9,Z 661.081,A -85,B 0,C 180,E1 -31653.324,E2 -31653.324} C_VEL
LIN {X 0,Y 64.872,Z 659.308,A -85,B 0,C 180,E1 -31657.36,E2 -31657.36} C_VEL
LIN {X 0,Y 64.987,Z 658.286,A -85,B 0,C 180,E1 -31661.072,E2 -31661.072} C_VEL
LIN {X 0,Y 64.994,Z 658.592,A -85,B 0,C 180,E1 -31662.744,E2 -31662.744} C_VEL
LIN {X 0,Y 64.932,Z 660.92,A -85,B 0,C 180,E1 -31666.275,E2 -31666.275} C_VEL
LIN {X 0,Y 64.932,Z 660.92,A -85,B 0,C 180,E1 -31666.275,E2 -31666.275}

QRS_NEXT_CUT()

QRS_NEXT()
QRS_HOME()

END
